(* CoDeSys 2.3.9.50 project: flat_v2.pro *)
(* Libraries: TcBABasic.lib 22.7.15 15:46:14, standard.lib 5.6.98 11:03:02, TcpIp.lib 9.1.14 13:33:22, TcBase.lib 14.5.09 11:14:08, TcSystem.lib 7.6.16 10:01:22, ModbusRTU.lib 13.5.15 12:38:16, TcIoFunctions.lib 27.1.17 16:22:22, COMlibV2.lb6 25.2.14 08:37:08, TcUtilities.lib 3.2.16 15:08:58 *)

(* Task configuration *)
TASK Standard (PRIORITY := 0, INTERVAL := T#50ms);
	MAIN
END_TASK

(* Global variable list: Global_Variables *)
VAR_GLOBAL


	Clear						: ClearComBuffer;
	MB							: ModbusRtuMaster_KL6x22B;
	TxBufferCom1				: ComBuffer;
	RxBufferCom1				: ComBuffer;
	SerialLineControlCom1			: SerialLineControl;
	ReceiveDataCom1			: ReceiveData;
	SendDataCom1				: SendData;
	Merc_address				: BYTE:=97;
	Sensor_CO2_high	 			: BYTE;	(*Старший байт датчика MH-Z19B*)
	Sensor_CO2_low 				: BYTE;	(*Младший байт датчика MH-Z19B*)
	iobroker						: iobroker_Struct;
	Modbus						: Modbus_Struct;
	Internal						: Internal_Struct;
(*
	MB_vars						: stMB;
	Mercury						: stMercury;
	iob_mqtt						: stIobroker;
*)
(*	Sensor_street_north_temp		: REAL;
	Sensor_sport_underfloor_temp	: REAL;
*)
	Sensor_control_temp			: WORD;
	Sensor_control_hum			: WORD;



	HW_temp_first_floor					AT %IW40:INT;	(* Датчик температуры 1 этаж *)
	HW_temp_second_floor				AT %IW42:INT;	(* Датчик температуры 2 этаж *)
	HW_temp_underfloor					AT %IW44:INT;	(* Датчик температуры подпол 1 этаж *)
	HW_temp_sport						AT %IW46:INT;	(* Датчик температуры спортзал *)

	HW_temp_sport_underfloor				AT %IW48:INT;	(* Датчик температуры подпол спортзал *)
	HW_temp_sauna						AT %IW50:INT;	(* Датчик температуры сауна*)
	HW_temp_street						AT %IW52:INT;	(* Датчик температуры улица *)
	HW_temp_vent						AT %IW54:INT;	(* Датчик температуры притока вентиляции *)

	HW_temp_balkon						AT %IW60:INT;	(* Датчик температуры  *)
	HW_temp_drovnik						AT %IW62:INT;	(* Датчик температуры *)
	HW_temp_sklad						AT %IW64:INT;	(* Датчик температуры  *)
	HW_temp_rezerv						AT %IW66:INT;	(* Датчик температуры  *)


	HW_PIR_terrasa						AT %IX56.0:BOOL;		(*PIR датчик терраса *)
	HW_PIR_zapad						AT %IX56.1:BOOL;		(*PIR датчик запад *)
	HW_PIR_vostok						AT %IX56.2:BOOL;		(*PIR датчик восток *)
	HW_PIR_sport						AT %IX56.3:BOOL;		(*PIR датчик спортзал *)

	HW_GERKON_drovnik					AT %IX56.4:BOOL;		(*Геркон дровник *)
	HW_GERKON_door					AT %IX56.5:BOOL;		(*Геркон дверь *)
	HW_sensor_smoke_1floor				AT %IX56.6:BOOL;		(*Датчик дыма 1 этаж *)
	HW_sensor_smoke_2_3floor			AT %IX56.7:BOOL;		(*Датчик дыма 2 этаж *)

	HW_button_light_garden				AT %IX57.0:BOOL;		(* Кнопка прожектор терраса  *)
	HW_sensor_smoke_sport				AT %IX57.1:BOOL;		(* Кнопка охрана  *)
	HW_button_vorota						AT %IX57.2:BOOL;		(* Кнопка открытия ворот  *)
	HW_button_kalitka					AT %IX57.3:BOOL;		(* Кнопка открытия калитки  *)

	HW_button_poliv_terrasa				AT %IX57.4:BOOL;		(* Кнопка полив терраса 2 часа  *)
	HW_button_poliv_zapad				AT %IX57.5:BOOL;		(* Кнопка полив запад  2 часа  *)
	HW_button_poliv_south				AT %IX57.6:BOOL;		(*  Кнопка полив юг  2 часа  *)
	HW_button_poliv_north					AT %IX57.7:BOOL;		(*  Кнопка полив север  2 часа  *)


	HW_sensor_supply					AT %IX58.0:BOOL;		(* Датчик напряжение  *)
	HW_GERKON_sklad					AT %IX58.1:BOOL;		(*Геркон *)
	HW_PIR_north_zapad					AT %IX58.2:BOOL;		(*PIR датчик  *)
	HW_PIR_north_vostok					AT %IX58.3:BOOL;		(*PIR датчик  *)


	HW_heat_first_floor					AT %QX0.0:BOOL;		(* Отопление 1 этаж *)
	HW_heat_second_floor				AT %QX0.1:BOOL;		(* Отопление 2 этаж *)
	HW_heat_sport						AT %QX0.2:BOOL;		(* Отопление спортзал *)
	HW_heat_underfloor					AT %QX0.3:BOOL;		(* Отопление подпол *)
	HW_heat_sauna						AT %QX0.4:BOOL;		(* Отопление сауна *)
	HW_heat_bathroom					AT %QX0.5:BOOL;		(* Отопление душевая *)
	HW_heat_pipe						AT %QX0.6:BOOL;		(* Отопление водопровод *)
	HW_vent_underfloor					AT %QX0.7:BOOL;		(* Вентиляция подпола *)

	HW_vorota							AT %QX1.0:BOOL;		(* Ворота *)
	HW_kalitka							AT %QX1.1:BOOL;		(* Калитка *)
	HW_pomp_house						AT %QX1.2:BOOL;		(* Насос водоснабжения дома *)
	HW_pomp_garden					AT %QX1.3:BOOL;		(* Насос полива *)
	HW_light_garden						AT %QX1.4:BOOL;		(* Прожектор двор *)
	HW_light_terrasa						AT %QX1.5:BOOL;		(* Свет терраса *)
	HW_light_rezerv						AT %QX1.6:BOOL;		(* Резервное освещение *)
	HW_switch_RS485					AT %QX1.7:BOOL:=TRUE;		(* RS485 line *)


	HW_vent_valve_input					AT %QX2.0:BOOL;		(* Клапан приточной вентиляции *)
	HW_vent_valve_output					AT %QX2.1:BOOL;		(* Клапан вытяжной вентиляции *)
	HW_trans_power						AT %QX2.2:BOOL;		(*Подача тока на трансформатор и реле ТЭН-а *)
	HW_vent_in_heat						AT %QX2.3:BOOL;		(* Подогрев притока - ТЭН *)
	HW_vent_in_heat_level				AT %QX2.4:BOOL;		(* Подогрев притока ночной режим   -5 К ТЭН *)
	HW_vent_in_trans_105_130				AT %QX2.5:BOOL:=FALSE;  (* Напряжение 110 или 130 В *)
	HW_vent_in_trans_160_220				AT %QX2.6:BOOL:=FALSE;  (* Напряжение 160 или 220 В *)
	HW_vent_in_trans_LO_HI				AT %QX2.7:BOOL:=FALSE;  (* Напряжение 110/130  или 160/220 В *)

	HW_poliv_terrasa						AT %QX3.0:BOOL;		(* полив терраса  *)
	HW_poliv_zapad						AT %QX3.1:BOOL;		(* полив запад   *)
	HW_poliv_south						AT %QX3.2:BOOL;		(* полив юг   *)
	HW_poliv_north						AT %QX3.3:BOOL;		(* полив север   *)
(*
	HW_level_light_1_floor					AT %QW4: WORD:=32767;	(* Уровень яркости света на 1 этаже *)
	HW_level_light_kitchen					AT %QW8: WORD:=32767;	(* Уровень яркости света на кухне *)
*)

END_VAR

(* Global variable list: TwinCAT_Configuration *)
(* Generated automatically by TwinCAT - (read only) *)
VAR_CONFIG
	MAIN.ToFromNovRam AT %QB56 : DataToFromNovram;	(*  ~ {LinkedWith:TIID^Device 2 (NOV/DP-RAM)^Outputs^Var4} *)
	.MB.InData AT %IB68 : MB_KL6inData22B;
	.MB.OutData AT %QB32 : MB_KL6outData22B;
END_VAR

(* Data type *)
TYPE DataToFromNovram :
STRUCT

	Target_CO2_mem					:		INT;
	First_floor_temp_target_mem		:		INT;
	Second_floor_temp_target_mem		:		INT;
	Sport_temp_target_mem			:		INT;
	Sauna_temp_target_mem			:		INT;
	Underfloor_temp_target_mem		:		INT;
	Underfloor_humidity_target_mem	:		INT;

	Pomp_house_mem				:		BOOL;
	Pomp_garden_mem				:		BOOL;

	Light_garden_mem				:		BOOL;

	Vent_mem						:		BOOL;
	Vent_heat_mem					:		INT;
	Vent_heat_level_mem				:		BOOL;

	Poliv_zapad_minutes				:		INT;
	Poliv_terrasa_minutes				:		INT;
	Poliv_south_minutes				:		INT;
	Poliv_north_minutes				:		INT;


END_STRUCT
END_TYPE

(* Data type *)
TYPE Internal_struct :
STRUCT
	Drovnik_temp					 :	REAL; 	(*12382*)			(* PT1000 *)
	Sklad_temp					 :	REAL; 	(*12384*)			(* PT1000 *)
	Rezerv_temp					 :	REAL; 	(*12386*)			(* PT1000 *)

	First_floor_temp 				:	REAL;	(*12288+100=12388*) (* PT1000 *)
	First_floor_hum 				:	REAL;	(*12390*)			(*SHT20		#1*)
	First_floor_CO2				:	REAL;	(*12392*)
	First_floor_temp_SHT20		:	REAL;	(*12394*)			(*SHT20		#1*)

	Second_floor_hum			:	REAL;	(*12396*)			(*SHT20		#2*)
	Second_floor_temp 			:	REAL;	(*12398*) 		(* PT1000 *)
	Second_floor_CO2 			:	REAL;	(*12400*)
	Sport_temp	 				:	REAL;	(*12402*)			(* PT1000 *)

	Sauna_temp	 				:	REAL;	(*12404*)			(* PT1000 *)
	Underfloor_temp				:	REAL;	(*12406*)			(* PT1000 *)
	Underfloor_hum				:	REAL;	(*12408*)			(*SHT20		#3*)
	Sport_underfloor_temp			:	REAL;	(*12410*)			(* PT1000 *)

	Sport_underfloor_hum			:	REAL;	(*12412*)			(*SHT20		#4*)
	Street_temp					:	REAL;	(*12414*)			(* PT1000 *)
	Vent_temp					:	REAL;	(*12416*)			(* PT1000 *)
	Sklad_temp_SHT20			:	REAL;	(*12418*)			(*SHT20		#5*)
	Sklad_hum					:	REAL;	(*12420*)			(*SHT20		#5*)
	Temp_vent_in				:	REAL;	(*12422*)			(* unused *)


	Uv1							:	REAL;	(*12424*)
	Uv2							:	REAL;	(*12426*)
	Uv3							:	REAL;	(*12428*)
	Pw1							:	REAL;	(*12430*)
	Pw2							:	REAL;	(*12432*)
	Pw3							:	REAL;	(*12434*)
	Pw_total						:	REAL;	(*12436*)
	Ia1							:	REAL;	(*12438*)
	Ia2							:	REAL;	(*12440*)
	Ia3							:	REAL;	(*12442*)
	E_T1						:	REAL;	(*12444*)
	E_T2						:	REAL; 	(*12288+158=12446*)

	Second_floor_temp_SHT20			:	REAL;	(*12448 *)		(*SHT20		#2*)
	Underfloor_temp_SHT20			:	REAL;	(*12450 *)		(*SHT20		#3*)
	Sport_underfloor_temp_SHT20		:	REAL;	(*12452 *)		(*SHT20		#4*)
	Street_temp_SHT20				:	REAL;	(*12454 *)		(*SHT20		#6*)
	Street_hum						:	REAL;	(*12456 *)		(*SHT20		#6*)

END_STRUCT
END_TYPE

(* Data type *)
TYPE iobroker_Struct  :
STRUCT
(*	Vent_status				: 	INT;
	Valve_status				: 	INT;
	First_floor_temp 			:	REAL;
	First_floor_temp_target 		:	INT;
	First_floor_hum 			:	REAL;
	First_floor_CO2			:	REAL;
	Kitchen_room_temp		:	REAL;
	Kitchen_room_hum		:	REAL;
	Second_floor_temp 		:	REAL;
	Second_floor_temp_target 	:	INT;
	Second_floor_CO2 		:	REAL;
	Sport_temp	 			:	REAL;
	Sport_temp_target			:	INT;
	Sauna_temp	 			:	REAL;
	Sauna_temp_target		:	INT;
	Underfloor_temp			:	REAL;
	Underfloor_temp_target	:	INT;
	Underfloor_humidity		:	REAL;
	Underfloor_humidity_target	:	INT;
	Sport_underfloor_temp		:	REAL;
	Sport_underfloor_hum		:	REAL;
	Street_temp				:	REAL;
	Vent_temp				:	REAL;
	Street_north_temp			:	REAL;
	Street_north_hum			:	REAL;
*)
	PIR_terrasa				:	BOOL:=TRUE;
	PIR_zapad				:	BOOL:=TRUE;
	PIR_vostok				:	BOOL:=TRUE;
	PIR_sport				:	BOOL:=TRUE;
	GERKON_drovnik			:	BOOL:=TRUE;
	Smoke					:	BOOL;
	Button_light_garden		:	BOOL;
	Light_garden				:	BOOL;
	Vorota_active				:	BOOL:=FALSE;
	Vorota_open_active		:	BOOL:=FALSE;
	Poliv_zapad				:	BOOL;
	Poliv_terrasa				:	BOOL;
	Poliv_south				:	BOOL;
	Poliv_north				:	BOOL;
(*
	Vent_input_level			:	INT;  (*  0-220 V  *)
	Vent_output_level			:	INT; (*0-100%*)
	Temp_vent_in			:	REAL;
	Vent_valve_status			:	INT;
	Security_status			:	BOOL;
	Target_CO2				:	INT;
	Vent						:	BOOL;
	Vent_underfloor			:	BOOL;
	Vent_out					:	BOOL;
	Vent_heat				:	INT;
	Vent_heat_level			:	BOOL;
	Vorota					:	BOOL;
	Vorota_open				:	BOOL;
	Kalitka					:	BOOL;
	
	Sensor_supply			:	BOOL;
	Pomp_house				:	BOOL;
	Pomp_garden			:	BOOL;
	Light_garden				:	BOOL;
	Poliv_zapad				:	BOOL;
	Poliv_terrasa				:	BOOL;
	Poliv_south				:	BOOL;
	Poliv_zapad_minutes		:	INT;
	Poliv_terrasa_minutes		:	INT;
	Poliv_south_minutes		:	INT;
	Uv1						:	REAL;
	Uv2						:	REAL;
	Uv3						:	REAL;
	Pw1						:	REAL;
	Pw2						:	REAL;
	Pw3						:	REAL;
	Pw_total					:	REAL;
	Ia1						:	REAL;
	Ia2						:	REAL;
	Ia3						:	REAL;
	E_T1					:	REAL;
	E_T2					:	REAL; (* 64 values*)
*)

(*	M1T1					:	DWORD:=0;
	M1T2					:	DWORD:=0; (* 66 values*)

	M2T1					:	DWORD:=0; (* 67 values*)
	M2T2					:	DWORD:=0;
	M3T1					:	DWORD:=0;
	M3T2					:	DWORD:=0;
	M4T1					:	DWORD:=0; (* 70 values*)
	M4T2					:	DWORD:=0;
	M5T1					:	DWORD:=0;
	M5T2					:	DWORD:=0;
	M6T1					:	DWORD:=0;
	M6T2					:	DWORD:=0;
	M7T1					:	DWORD:=0;
	M7T2					:	DWORD:=0;
	M8T1					:	DWORD:=0;
	M8T2					:	DWORD:=0;
	M9T1					:	DWORD:=0;
	M9T2					:	DWORD:=0;
	M10T1					:	DWORD:=0;
	M10T2					:	DWORD:=0;
	M11T1					:	DWORD:=0;
	M11T2					:	DWORD:=0;
	M12T1					:	DWORD:=0;
	M12T2					:	DWORD:=0;   (* 86 values*)
*)

END_STRUCT
END_TYPE

(* Data type *)
TYPE Modbus_struct :
STRUCT
	Vent_status					AT %MB100	:	INT;		(*12288+50=12338*)
	Valve_status					AT %MB102	: 	INT;		(*12339*)
	First_floor_temp_target 			AT %MB104	:	INT;		(*12340*)
	Second_floor_temp_target 		AT %MB106	:	INT;		(*12341*)
	Sport_temp_target				AT %MB108	:	INT;		(*12342*)
	Sauna_temp_target			AT %MB110	:	INT;		(*12343*)
	Underfloor_temp_target		AT %MB112	:	INT;		(*12344*)
	Underfloor_humidity_target		AT %MB114	:	INT;		(*12345*)
	PIR_terrasa					AT %MB116	:	BOOL:=TRUE;	(*12346*)
	PIR_zapad					AT %MB118	:	BOOL:=TRUE;	(*12347*)
	PIR_vostok					AT %MB120	:	BOOL:=TRUE;	(*12348*)
	PIR_sport					AT %MB122	:	BOOL:=TRUE;	(*12349*)
	GERKON_drovnik				AT %MB124	:	BOOL:=TRUE;	(*12288+62=12350*)

	Vent_input_level				AT %MB126	:	INT; 			 (*12351			*  0-220 V  *)
	Vent_output_level				AT %MB128	:	INT; 			(*12352			0-100%*)
	Vent_valve_status				AT %MB130	:	INT;		(*12353*)
	Target_CO2					AT %MB132	:	INT;		(*12354*)
	Security_status				AT %MB134	:	BOOL;	(*12355*)
	Vent							AT %MB136	:	BOOL;	(*12356*)
	Vent_underfloor				AT %MB138	:	BOOL;	(*12357*)
	Vent_out						AT %MB140	:	BOOL;	(*12358*)
	Vent_heat					AT %MB142	:	INT;		(*12359*)
	Vent_heat_level				AT %MB144	:	BOOL;	(*12360*)
	Vorota						AT %MB146	:	BOOL;	(*12361*)
	Vorota_open					AT %MB148	:	BOOL;	(*12362*)
	Kalitka						AT %MB150	:	BOOL;	(*12363*)
(*
	Smoke						AT %MB152	:	BOOL;	(*12364*)
*)
	Sensor_supply				AT %MB154	:	BOOL;	(*12365*)
	Pomp_house					AT %MB156	:	BOOL;	(*12366*)
	Pomp_garden				AT %MB158	:	BOOL;	(*12367*)
	Light_garden					AT %MB160	:	BOOL;	(*12368*)
	Poliv_zapad					AT %MB162	:	BOOL;	(*12369*)
	Poliv_terrasa					AT %MB164	:	BOOL;	(*12370*)
	Poliv_south					AT %MB166	:	BOOL;	(*12371*)
	Poliv_zapad_minutes			AT %MB168	:	INT;		(*12372*)
	Poliv_terrasa_minutes			AT %MB170	:	INT;		(*12373*)
	Poliv_south_minutes			AT %MB172	:	INT;		(*12288 +86=  12374*)
	Poliv_north_minutes			AT %MB174	:	INT	;	(*12375 *)
	Poliv_north					AT %MB176	:	BOOL;	(*12376*)






	Drovnik_temp					AT %MW188 :	REAL; 	(*12382*)			(* PT1000 *)
	Sklad_temp					AT %MW192 :	REAL; 	(*12384*)			(* PT1000 *)
	Rezerv_temp					AT %MW196 :	REAL; 	(*12386*)			(* PT1000 *)

	First_floor_temp 				AT %MW200	:	REAL;	(*12288+100=12388*) (* PT1000 *)
	First_floor_hum 				AT %MW204	:	REAL;	(*12390*)			(*SHT20		#1*)
	First_floor_CO2				AT %MW208	:	REAL;	(*12392*)
	First_floor_temp_SHT20		AT %MW212	:	REAL;	(*12394*)			(*SHT20		#1*)

	Second_floor_hum			AT %MW216	:	REAL;	(*12396*)			(*SHT20		#2*)
	Second_floor_temp 			AT %MW220	:	REAL;	(*12398*) 		(* PT1000 *)
	Second_floor_CO2 			AT %MW224	:	REAL;	(*12400*)
	Sport_temp	 				AT %MW228	:	REAL;	(*12402*)			(* PT1000 *)

	Sauna_temp	 				AT %MW232	:	REAL;	(*12404*)			(* PT1000 *)
	Underfloor_temp				AT %MW236	:	REAL;	(*12406*)			(* PT1000 *)
	Underfloor_hum				AT %MW240	:	REAL;	(*12408*)			(*SHT20		#3*)
	Sport_underfloor_temp			AT %MW244	:	REAL;	(*12410*)			(* PT1000 *)

	Sport_underfloor_hum			AT %MW248	:	REAL;	(*12412*)			(*SHT20		#4*)
	Street_temp					AT %MW252	:	REAL;	(*12414*)			(* PT1000 *)
	Vent_temp					AT %MW256	:	REAL;	(*12416*)			(* PT1000 *)
	Sklad_temp_SHT20			AT %MW260	:	REAL;	(*12418*)			(*SHT20		#5*)
	Sklad_hum					AT %MW264	:	REAL;	(*12420*)			(*SHT20		#5*)
	Temp_vent_in				AT %MW268	:	REAL;	(*12422*)			(* unused *)


	Uv1							AT %MW272	:	REAL;	(*12424*)
	Uv2							AT %MW276	:	REAL;	(*12426*)
	Uv3							AT %MW280	:	REAL;	(*12428*)
	Pw1							AT %MW284	:	REAL;	(*12430*)
	Pw2							AT %MW288	:	REAL;	(*12432*)
	Pw3							AT %MW292	:	REAL;	(*12434*)
	Pw_total						AT %MW296	:	REAL;	(*12436*)
	Ia1							AT %MW300	:	REAL;	(*12438*)
	Ia2							AT %MW304	:	REAL;	(*12440*)
	Ia3							AT %MW308	:	REAL;	(*12442*)
	E_T1						AT %MW312	:	REAL;	(*12444*)
	E_T2						AT %MW316	:	REAL; 	(*12288+158=12446*)

	Second_floor_temp_SHT20		AT %MW320	:	REAL;	(*12448 *)		(*SHT20		#2*)
	Underfloor_temp_SHT20		AT %MW324	:	REAL;	(*12450 *)		(*SHT20		#3*)
	Sport_underfloor_temp_SHT20	AT %MW328	:	REAL;	(*12452 *)		(*SHT20		#4*)
	Street_temp_SHT20			AT %MW332	:	REAL;	(*12454 *)		(*SHT20		#6*)
	Street_hum					AT %MW336	:	REAL;	(*12456 *)		(*SHT20		#6*)


	Smoke_1floor					AT %MB400	:	BOOL;	(*12288+200=12488*)
	Smoke_2_3floor				AT %MB402	:	BOOL;	(*12489*)
	Smoke_sport					AT %MB404	:	BOOL;	(*12490*)
	Rezerv_2					AT %MB406	:	BOOL;	(*12491*)
	PIR_north_zapad				AT %MB408	:	BOOL;	(*12492*)
	PIR_north_vostok				AT %MB410	:	BOOL;	(*12493*)
	Gerkon_sklad				AT %MB412	:	BOOL;	(*12494*)
	Gerkon_door					AT %MB414	:	BOOL;	(*12495*)
	Light_reserv					AT %MB416	:	BOOL;	(*12496*)
	Light_reserv_manual			AT %MB418	:	INT;		(*12497*)
	Supply_akb					AT %MB420	:	REAL;	(*12498*)
	Security_delay				AT %MB424	:	INT;		(*12500*)
	Balkon_temp					AT %MW428 :	REAL; 	(*12502*)			(* PT1000 *)

	Poliv_zapad_minutes_est		AT %MB500	:	INT;		(*12288+250=12538*)
	Poliv_terrasa_minutes_est		AT %MB502	:	INT;		(*12539*)
	Poliv_south_minutes_est		AT %MB504	:	INT;		(*12540*)
	Poliv_north_minutes_est		AT %MB506	:	INT	;	(*12541 *)

	Kitchen_room_CO2			AT %MB508	:	INT;

	M1T1					AT %MB600	:	REAL;
	M1T2					AT %MB604	:	REAL;
	M2T1					AT %MB608	:	REAL;
	M2T2					AT %MB612	:	REAL;
	M3T1					AT %MB616	:	REAL;
	M3T2					AT %MB620	:	REAL;
	M4T1					AT %MB624	:	REAL;
	M4T2					AT %MB628	:	REAL;
	M5T1					AT %MB632	:	REAL;
	M5T2					AT %MB636	:	REAL;
	M6T1					AT %MB640	:	REAL;
	M6T2					AT %MB644	:	REAL;
	M7T1					AT %MB648	:	REAL;
	M7T2					AT %MB652	:	REAL;
	M8T1					AT %MB656	:	REAL;
	M8T2					AT %MB660	:	REAL;
	M9T1					AT %MB664	:	REAL;
	M9T2					AT %MB668	:	REAL;
	M10T1					AT %MB672	:	REAL;
	M10T2					AT %MB676	:	REAL;
	M11T1					AT %MB680	:	REAL;
	M11T2					AT %MB684	:	REAL;
	M12T1					AT %MB688	:	REAL;
	M12T2					AT %MB692	:	REAL;


END_STRUCT
END_TYPE

(* Data type *)
(* @NESTEDCOMMENTS := 'Yes' *)
(* @PATH := '' *)
(* @OBJECTFLAGS := '0, 8' *)
TYPE ST_MqttReceivedPublishTelegram :
STRUCT
	sTopic		: STRING[255];
	sValue		: STRING[255];
	bHasData	: BOOL;
END_STRUCT
END_TYPE
(* @END_DECLARATION := '0' *)

(* Data type *)
(* @NESTEDCOMMENTS := 'Yes' *)
(* @PATH := '' *)
(* @OBJECTFLAGS := '0, 8' *)
TYPE ST_MqttSettings :
STRUCT
	(* informations *)
	sMqttClientId	: STRING[23];
	sMqttUserId	: STRING[25];
	sMqttPassword	: STRING[25];
	sMqttBrokerIP	: STRING[15];
	nMqttBrokerPort	: UDINT := 1883;

	(* state *)
	bSocketConnection	: BOOL := FALSE;
	bConnected			: BOOL := FALSE;
	bConnectPackageSent	: BOOL := FALSE;
	bDisconnect			: BOOL := FALSE;
	bError				: BOOL := FALSE;
	bValidConnection	: BOOL := FALSE;
	bActive				: BOOL := FALSE;
	wPackageIdentifier	: WORD := 1;
	hSocket				: T_HSOCKET;
	tonSendPingReq		: TON;

	(* send *)
	stMqttSendTelegram			: ST_MqttTelegram;
	stMqttLastSendTelegram		: ST_MqttTelegram;

	(* receive *)
	stMqttReceivedTelegram			: ST_MqttTelegram;
	stMqttLastReceivedTelegram		: ST_MqttTelegram;
	stMqttReceivedPublishTelegram	: ST_MqttReceivedPublishTelegram;

	(* settings internal *)
	iTelegramSize	: INT := 544;
	usKeepAliveTime	: USINT := 60; (* seconds *)

END_STRUCT
END_TYPE
(* @END_DECLARATION := '0' *)

(* Data type *)
(* @NESTEDCOMMENTS := 'Yes' *)
(* @PATH := '' *)
(* @OBJECTFLAGS := '0, 8' *)
TYPE ST_MqttTelegram :
STRUCT
	arMqttData 	: ARRAY[0..544] OF BYTE;
	nDataLength	: UDINT := 0;
END_STRUCT
END_TYPE
(* @END_DECLARATION := '0' *

(* Data type *)
TYPE stIobroker :
STRUCT

	Control_hum					:	REAL;
	Control_temp					:	REAL;
	Control_hum2					:	REAL;
	Control_temp2				:	REAL;

END_STRUCT
END_TYPE

(* Data type *)
TYPE stMB :
STRUCT

	M1T1							AT %MW0	:REAL;  	(* modbus address 12288 *)
	M1T2							AT %MW4	:REAL;	(* 12290 *)
	M2T1							AT %MW8	:REAL;	(* 12292 *)
	M2T2							AT %MW12	:REAL;	 (* 12294 *)
	M3T1							AT %MW16	:REAL;	 (* 12296 *)
	M3T2							AT %MW20	:REAL;	 (* 12298 *)
	M4T1							AT %MW24	:REAL;	 (* 12300 *)
	M4T2							AT %MW28	:REAL;	 (* 12302 *)
	M5T1							AT %MW32	:REAL;	 (* 12304 *)
	M5T2							AT %MW36	:REAL;	 (* 12306 *)
	M6T1							AT %MW40	:REAL;	 (* 12308 *)
	M6T2							AT %MW44	:REAL;	(* 12310 *)
	M7T1							AT %MW48	:REAL;	 (* 12312 *)
	M7T2							AT %MW52	:REAL;	 (* 12314 *)
	M8T1							AT %MW56	:REAL;	 (* 12316 *)
	M8T2							AT %MW60	:REAL;	(* 12318 *)
	M9T1							AT %MW64	:REAL;	(* 12320 *)
	M9T2							AT %MW68	:REAL;	(* 12322 *)
	M10T1							AT %MW72	:REAL;	(* 12324 *)
	M10T2							AT %MW76	:REAL;	(* 12326 *)
	M11T1							AT %MW80	:REAL;	(* 12328 *)
	M11T2							AT %MW84	:REAL;	(* 12330 *)
	M12T1							AT %MW88	:REAL;	(* 12332 *)
	M12T2							AT %MW92	:REAL;	(* 12334 *)

END_STRUCT
END_TYPE

(* Data type *)
TYPE stMercury :
STRUCT

	M1T1					:	REAL;
	M1T2					:	REAL;
	M2T1					:	REAL;
	M2T2					:	REAL;
	M3T1					:	REAL;
	M3T2					:	REAL;
	M4T1					:	REAL;
	M4T2					:	REAL;
	M5T1					:	REAL;
	M5T2					:	REAL;
	M6T1					:	REAL;
	M6T2					:	REAL;
	M7T1					:	REAL;
	M7T2					:	REAL;
	M8T1					:	REAL;
	M8T2					:	REAL;
	M9T1					:	REAL;
	M9T2					:	REAL;
	M10T1					:	REAL;
	M10T2					:	REAL;
	M11T1					:	REAL;
	M11T2					:	REAL;
	M12T1					:	REAL;
	M12T2					:	REAL;

END_STRUCT
END_TYPE

(* POU MAIN, ST *)
PROGRAM MAIN
VAR
	ToFromNovRam			AT %Q*:DataToFromNovram;
	INITVAR					: BOOL:=FALSE;




END_VAR
IF (INITVAR=FALSE) THEN

	(* START RESTORE VARS FROM MEMORY AFTER REBOOT/RESET/LOST POWER *)

	Modbus.Target_CO2				:=	ToFromNovRam.Target_CO2_mem;
	Modbus.First_floor_temp_target		:=	ToFromNovRam.First_floor_temp_target_mem;
	Modbus.Second_floor_temp_target	:=	ToFromNovRam.Second_floor_temp_target_mem;
	Modbus.Sport_temp_target			:=	ToFromNovRam.Sport_temp_target_mem;
	Modbus.Sauna_temp_target		:=	ToFromNovRam.Sauna_temp_target_mem;

	Modbus.Underfloor_temp_target		:=	ToFromNovRam.Underfloor_temp_target_mem;
	Modbus.Underfloor_humidity_target	:=	ToFromNovRam.Underfloor_humidity_target_mem;

	Modbus.Vent						:=	ToFromNovRam.Vent_mem;
	Modbus.Vent_heat				:=	ToFromNovRam.Vent_heat_mem;
	Modbus.Vent_heat_level			:=	ToFromNovRam.Vent_heat_level_mem;

	Modbus.Pomp_house				:=	ToFromNovRam.Pomp_house_mem;
	Modbus.Pomp_garden				:=	ToFromNovRam.Pomp_garden_mem;
	Modbus.Light_garden				:=	ToFromNovRam.Light_garden_mem;

	Modbus.Poliv_zapad_minutes		:=	ToFromNovRam.Poliv_zapad_minutes;
	Modbus.Poliv_terrasa_minutes		:=	ToFromNovRam.Poliv_terrasa_minutes;
	Modbus.Poliv_south_minutes		:=	ToFromNovRam.Poliv_south_minutes;
	Modbus.Poliv_north_minutes		:=	ToFromNovRam.Poliv_north_minutes;

	(* END RESTORE VARS FROM MEMORY AFTER REBOOT/RESET/LOST POWER *)

	INITVAR:=TRUE;
ELSE
	(*START SAVE VARS to PERSISTENT MEMORY*)
	ToFromNovRam.Target_CO2_mem					:=	Modbus.Target_CO2;
	ToFromNovRam.First_floor_temp_target_mem			:=	Modbus.First_floor_temp_target;
	ToFromNovRam.Second_floor_temp_target_mem		:=	Modbus.Second_floor_temp_target;
	ToFromNovRam.Sport_temp_target_mem			:=	Modbus.Sport_temp_target;
	ToFromNovRam.Sauna_temp_target_mem			:=	Modbus.Sauna_temp_target;

	ToFromNovRam.Underfloor_temp_target_mem		:=	Modbus.Underfloor_temp_target;
	ToFromNovRam.Underfloor_humidity_target_mem		:=	Modbus.Underfloor_humidity_target;

	ToFromNovRam.Vent_mem						:=	Modbus.Vent;
	ToFromNovRam.Vent_heat_mem					:=	Modbus.Vent_heat;
	ToFromNovRam.Vent_heat_level_mem				:=	Modbus.Vent_heat_level;

	ToFromNovRam.Pomp_house_mem				:=	Modbus.Pomp_house;
	ToFromNovRam.Pomp_garden_mem			:=	Modbus.Pomp_garden;
	ToFromNovRam.Light_garden_mem				:=	Modbus.Light_garden;


	ToFromNovRam.Poliv_zapad_minutes			:=	Modbus.Poliv_zapad_minutes;
	ToFromNovRam.Poliv_terrasa_minutes			:=	Modbus.Poliv_terrasa_minutes;
	ToFromNovRam.Poliv_south_minutes			:=	Modbus.Poliv_south_minutes;
	ToFromNovRam.Poliv_north_minutes			:=	Modbus.Poliv_north_minutes;

	(*END SAVE VARS to PERSISTENT MEMORY*)


	Sensors;						(* Аналогвые датчики на шине KL *)
	Security_new;						(* Мониторинг датчиков охраны *)
	RS485read;					(* Опрос устройств на шине RS485 *)
(*	Mqtt;	*)					(* MQTT *)
	Thermocontrol;				(* Термостат*)
	VentControl;					(* Глобальный контроль вентустановки*)
	VentPower;					(* Авторегулировка мощности вентустановки по датчикам CO2*)
	Poliv;						(* Таймеры зонального полива *)
	Power_act;					(*Контроль резервного освещения*)



(* Прямое присовение виртуальных переменных к переменным, жестко привязаным к физ. портам. Частота обновления= циклу ПЛК (50 мсек) : *)
	HW_pomp_house				:=	Modbus.Pomp_house;
	Modbus.Sensor_supply		:=	HW_sensor_supply;
	HW_vent_underfloor			:=	Modbus.Vent_underfloor;

	HW_kalitka					:=	Modbus.Kalitka;
	iobroker.button_light_garden	:=	HW_button_light_garden;
	HW_light_garden				:=	Modbus.Light_garden;
	iobroker.Light_garden			:=	Modbus.Light_garden;


	Buttons;						(*Обработка нажатия кнопок *)

END_IF
END_PROGRAM

(* POU Sensors, ST *)
PROGRAM Sensors
VAR
(*	Period_sensors_read		: INT:=30; *) (* Частота присвоения значений аналоговых температурных датчиков с модулей KL, секунды *)
	Timer					: TON;
	TimerQ					: BOOL;
	tTimerValue				: TIME:=t#30s; (* Частота присвоения значений аналоговых температурных датчиков с модулей KL, секунды *)
END_VAR
Timer();

(* tTimerValue := DINT_TO_TIME(Period_sensors_read*1000); *)

	Timer(IN:=NOT TimerQ , PT:=tTimerValue , Q=>TimerQ , ET=> );
	IF timer.q THEN

		Modbus.First_floor_temp		:=	INT_TO_REAL(HW_temp_first_floor)/10;
		Modbus.Second_floor_temp	:=	INT_TO_REAL(HW_temp_second_floor)/10;
		Modbus.Sauna_temp			:=	INT_TO_REAL(HW_temp_sauna)/10;
		Modbus.Sport_temp			:=	INT_TO_REAL(HW_temp_sport)/10;

		Modbus.Underfloor_temp		:=	INT_TO_REAL(HW_temp_underfloor)/10;
		Modbus.Sport_underfloor_temp	:=	INT_TO_REAL(HW_temp_sport_underfloor)/10;
		Modbus.Street_temp			:=	INT_TO_REAL(HW_temp_street)/10;
		Modbus.Vent_temp			:=	INT_TO_REAL(HW_temp_vent)/10;

		Modbus.Balkon_temp			:=	INT_TO_REAL(HW_temp_balkon)/10;
		Modbus.Drovnik_temp			:=	INT_TO_REAL(HW_temp_drovnik)/10;
		Modbus.Sklad_temp			:= 	INT_TO_REAL(HW_temp_sklad)/10;

	END_IF
END_PROGRAM

(* POU Security_new, ST *)
PROGRAM Security_new
VAR
(*	TRIG_PIR_terrasa			:	F_TRIG;
	TRIG_PIR_zapad			:	F_TRIG;
	TRIG_PIR_vostok			:	F_TRIG;
	TRIG_PIR_sport			:	F_TRIG;
	TRIG_GERKON_drovnik	:	F_TRIG;
	TRIG_sensor_smoke_1floor:	F_TRIG;

	trig_mem_terrasa				:	BOOL:=FALSE;
	trig_mem_zapad				:	BOOL:=FALSE;
	trig_mem_vostok				:	BOOL:=FALSE;
	trig_mem_sport				:	BOOL:=FALSE;
	trig_mem_drovnik				:	BOOL:=FALSE;
	trig_mem_sensor_smoke_1floor	:	BOOL:=FALSE;
*)
END_VAR
iobroker.PIR_terrasa			 :=HW_PIR_terrasa;
iobroker.PIR_zapad			 :=HW_PIR_zapad;
iobroker.PIR_vostok 			 :=HW_PIR_vostok;
iobroker.PIR_sport			 :=HW_PIR_sport;
iobroker.GERKON_drovnik		 :=HW_GERKON_drovnik;

Modbus.Smoke_1floor				 :=HW_sensor_smoke_1floor;
Modbus.Smoke_2_3floor			 :=HW_sensor_smoke_2_3floor;
Modbus.Smoke_sport				 :=HW_sensor_smoke_sport;


Modbus.PIR_terrasa			 :=HW_PIR_terrasa;
Modbus.PIR_zapad			 :=HW_PIR_zapad;
Modbus.PIR_vostok 			 :=HW_PIR_vostok;
Modbus.PIR_sport				 :=HW_PIR_sport;
Modbus.PIR_north_zapad		 :=HW_PIR_north_zapad;
Modbus.PIR_north_vostok		 :=HW_PIR_north_vostok;

Modbus.GERKON_door		 :=HW_GERKON_door;
Modbus.GERKON_drovnik		 :=HW_GERKON_drovnik;
Modbus.GERKON_sklad		 :=HW_GERKON_sklad;



(* Modbus.Smoke				 :=HW_sensor_smoke_1floor; *)
END_PROGRAM

(* POU RS485read, ST *)
PROGRAM RS485read
VAR
(*	Period_vent_switch	: INT:=180; *)
	CO2_period			: TIME;
	tTimerValue			: TIME	:=	t#180s; (* Период опроса RS485*)

	password_1				: ARRAY [1..6] OF BYTE:=6(1); (* пароль к меркуриям, по умолчанию 6 единиц*)
	crctest					: WORD;
	arrReceive				: ARRAY[1..22] OF BYTE;
	arrSend					: ARRAY[1..22] OF BYTE;

	MBdata					 : ARRAY [1..2] OF INT;
	FtrigBusy				: F_TRIG;
	timeoutvalue				: TIME := T#1000ms;		(* timeout while waiting for an answer of the modbus slave *)
	state					: INT;
	busy					: BOOL;
	LastErrorstate				: INT;
	LastModbusError			: ST_ModbusErrorDiagnostics;
	CounterError				: DINT;
	CounterSuccess			: DINT;
	Timer1					: TON;
	Timer1Q					: BOOL;
	Timer_day				:TON;
	Timer_dayQ				:BOOL;
	Timer_CO2				:TON;
(*	Timer_CO2Q				:BOOL; *)

	tmCheck					:TON;
	i,k,l,m,t					: INT:=1;


	sensors_SHT20_v1_id			: ARRAY[1..2] OF BYTE:=16#05, 16#0F;
	sensors_SHT20_v1_hum		: ARRAY[1..2] OF REAL:=2(0);
	sensors_SHT20_v1_temp		: ARRAY[1..2] OF REAL:=2(0);

	sensors_SHT20_v2_id			: ARRAY[1..4] OF BYTE:= 16#07, 16#08, 16#09,16#0A;
	sensors_SHT20_v2_hum		: ARRAY[1..4] OF REAL:=4(0);
	sensors_SHT20_v2_temp		: ARRAY[1..4] OF REAL:=4(0);


	sensors_CO2_id				: ARRAY[1..1] OF BYTE:=16#68;
	sensors_CO2_ppm			: ARRAY[1..1] OF INT;

	energyMT					: ARRAY[1..12,1..2] OF REAL;

	get_co2_mh_z19b_1floor	: FB_GET_CO2_MH_Z19B;
	get_co2_mh_z19b_2floor	: FB_GET_CO2_MH_Z19B;
	get_supply				: FB_GET_SUPPLY;
	get_current				: FB_GET_CURRENT;
	get_power				: FB_GET_POWER;
	get_energy_E_T1			: FB_GET_ENERGY;
	get_energy_E_T2			: FB_GET_ENERGY;

	get_energy_MT			: FB_GET_ENERGY;



	get_co2_mh_z19b_1floor_done	: BOOL;
	get_co2_mh_z19b_2floor_done	: BOOL;
	get_supply_done			: BOOL;
	get_current_done			: BOOL;
	get_power_done			: BOOL;

	get_energy_E_T1_done	: BOOL;
	get_energy_E_T2_done	: BOOL;
	get_energy_MT_done		: BOOL;

END_VAR
tmCheck();
Timer_day();
Timer_CO2();


IF (Modbus.Security_status = TRUE) THEN
	CO2_period	:= T#30m;
ELSE
	CO2_period 	:= T#2m;
END_IF


CASE state OF
	0:
		MB.ReadRegs(Execute:= FALSE);
		state := 1;


1:
	Clear(Buffer := RxBufferCom1);
		MB.ReadRegs(
			UnitID:= sensors_SHT20_v1_id[i],
			Quantity:= 2,
			MBAddr:= 0,
			cbLength:= 6,
			pMemoryAddr:= ADR(MBdata),
			Execute:= TRUE,
			Timeout:= timeoutvalue,
			Busy => busy,
		);
		IF NOT busy THEN
			IF (mb.Error = FALSE ) THEN
				sensors_SHT20_v1_temp[i]:=INT_TO_REAL(MBdata[1])/10;
				sensors_SHT20_v1_hum[i]:=INT_TO_REAL(MBdata[2])/10;
			END_IF
			i:=i+1;
			MB.ReadRegs(Execute:= FALSE);
			IF (i>2 )	THEN
				i:=1;
				Internal.First_floor_temp_SHT20		:=	sensors_SHT20_v1_temp[1];
				Internal.First_floor_hum				:=	sensors_SHT20_v1_hum[1];
				Internal.Street_temp_SHT20			:=	sensors_SHT20_v1_temp[2];
				Internal.Street_hum				:=	sensors_SHT20_v1_hum[2];
				Modbus.First_floor_temp_SHT20	:=	(sensors_SHT20_v1_temp[1]);
				Modbus.First_floor_hum			:=	(sensors_SHT20_v1_hum[1]);
				Modbus.Street_temp_SHT20		:=	(sensors_SHT20_v1_temp[2]);
				Modbus.Street_hum				:=	(sensors_SHT20_v1_hum[2]);
				state :=2;
			ELSE
				state :=1;
			END_IF

		END_IF

2:

		MB.ReadInputRegs(
			UnitID:= sensors_SHT20_v2_id[l],
			Quantity:= 2,
			MBAddr:= 1,
			cbLength:= 6,
			pMemoryAddr:= ADR(MBdata),
			Execute:= TRUE,
			Timeout:= timeoutvalue,
			Busy => busy,
		);
		IF NOT busy THEN
			IF (mb.Error = FALSE ) THEN
				sensors_SHT20_v1_temp[l]:=INT_TO_REAL(MBdata[1])/10;
				sensors_SHT20_v1_hum[l]:=INT_TO_REAL(MBdata[2])/10;
			END_IF
			l:=l+1;
			MB.ReadRegs(Execute:= FALSE);
			IF (l>4 )	THEN
				l:=1;
				Internal.Underfloor_temp_SHT20				:=	sensors_SHT20_v2_temp[1];
				Internal.Underfloor_hum					:=	sensors_SHT20_v2_hum[1];
				Internal.Sport_underfloor_temp_SHT20		:=	sensors_SHT20_v2_temp[2];
				Internal.Sport_underfloor_hum				:=	sensors_SHT20_v2_hum[2];
				Internal.Second_floor_temp_SHT20			:=	sensors_SHT20_v2_temp[3];
				Internal.Second_floor_hum					:=	sensors_SHT20_v2_hum[3];
				Internal.Sklad_temp_SHT20					:=	sensors_SHT20_v2_temp[4];
				Internal.Sklad_hum						:=	sensors_SHT20_v2_hum[4];


				Modbus.Underfloor_temp_SHT20			:=	(sensors_SHT20_v2_temp[1]);
				Modbus.Underfloor_hum					:=	(sensors_SHT20_v2_hum[1]);
				Modbus.Sport_underfloor_temp_SHT20		:=	(sensors_SHT20_v2_temp[2]);
				Modbus.Sport_underfloor_hum				:=	(sensors_SHT20_v2_hum[2]);
				Internal.Second_floor_temp_SHT20			:=	sensors_SHT20_v2_temp[3];
				Internal.Second_floor_hum					:=	sensors_SHT20_v2_hum[3];
				Internal.Sklad_temp_SHT20					:=	sensors_SHT20_v2_temp[4];
				Internal.Sklad_hum						:=	sensors_SHT20_v2_hum[4];

				state :=3;
			ELSE
				state :=2;
			END_IF

		END_IF



3:
		MB.ReadInputRegs(
			UnitID:=sensors_CO2_id[k], (* station address *)
			Quantity:= 1,
			MBAddr:= 3,
			cbLength:= 4,
			pMemoryAddr:= ADR(MBdata),
			Execute:= TRUE,
			Timeout:= timeoutvalue,
			Busy => busy	);
		IF NOT busy THEN
			IF (mb.Error = FALSE ) THEN
				sensors_CO2_ppm[k]	:=	(MBdata[1]);
			END_IF
			k:=k+1;
			MB.ReadRegs(Execute:= FALSE);
			IF (k>1 )	THEN
				k:=1;

				Modbus.Kitchen_room_CO2		:=	(sensors_CO2_ppm[1]);

				state :=5;
			ELSE
				state :=3;
			END_IF
		END_IF


5:

		tmCheck(in:=FALSE);
		tmCheck(in:=TRUE,pt:=t#2s);
		get_co2_mh_z19b_2floor_done := FALSE;
		get_co2_mh_z19b_2floor( co2=>Modbus.Second_Floor_CO2, done=>get_co2_mh_z19b_2floor_done);
		IF get_co2_mh_z19b_2floor_done = TRUE THEN
			state:=105;
		ELSIF tmcheck.Q THEN
			 state:=105;
		END_IF


105: (*открываем канал*)


	Clear(Buffer := RxBufferCom1);
	arrSend[1]:=Merc_address;
	arrSend[2]:=1; (*код доступа*)
	arrSend[3]:=1; (*Уровень доступа*)

	MEMCPY(ADR(arrSend)+3,ADR(password_1),6); (*пароль*)
	crctest:=F_CRC16(ADR(arrSend),9); (*расчет контрольной суммы*)
	MEMCPY(ADR(arrSend)+9,ADR(crctest),SIZEOF(crctest)); (*прибавление контрольной суммы к запросу*)
	SendDataCom1(pSendData:=ADR(arrSend),Length:=11,TXBuffer:=TxBufferCom1,Busy=>,Error=>);
	tmCheck(in:=FALSE); tmCheck(in:=TRUE,pt:=t#2s); 	(*запуск таймера проверки - потеря связи\обрыв кабеля*)
	state:=106;

106: (*ответ*)
	ReceiveDataCom1(pPrefix:=,LenPrefix:=,pSuffix:=,LenSuffix:=,
	pReceiveData:=ADR(arrReceive),SizeReceiveData:=4,
	Timeout:=t#2s,Reset:=,
	RXbuffer:=RxBufferCom1,
	DataReceived=>,busy=>,Error=>,RxTimeout=>,LenReceiveData=>);
	IF ReceiveDataCom1.Error <> 0 THEN
		state:=888;
	END_IF
	IF receiveDataCom1.DataReceived THEN
		state:=107;
	ELSIF tmcheck.Q THEN
		state:=888;
	END_IF
107: (*проверка ответа*)

	IF arrReceive[1] = Merc_address THEN
		state:= 108;
	ELSE
		state:=888;
	END_IF



108:
		tmCheck(in:=FALSE);
		tmCheck(in:=TRUE,pt:=t#2s);
		get_supply_done := FALSE;
		get_supply( byte1:=16#8, byte2:=16#16, byte3:=16#11,  supply1=>Modbus.UV1,supply2=>Modbus.UV2,supply3=>Modbus.UV3, done=>get_supply_done);
		IF get_supply_done = TRUE THEN
			state:=109;
		ELSIF tmcheck.Q THEN
			 state:=888;
		END_IF

 (*запрос на чтение тока  на всех фазах
--------------------------------------------------------------------------------------------------------------------------------------------------------------------
*)
109:
		tmCheck(in:=FALSE);
		tmCheck(in:=TRUE,pt:=t#2s);
		get_current_done := FALSE;
		get_current(byte1:=16#8, byte2:=16#16, byte3:=16#21,  current1=>Modbus.Ia1,current2=>Modbus.Ia2,current3=>Modbus.Ia3, done=>get_current_done);
		IF get_current_done = TRUE THEN
			state:=110;
		ELSIF tmcheck.Q THEN state:=888;
		END_IF

 (*запрос на чтение мощности  на всех фазах
--------------------------------------------------------------------------------------------------------------------------------------------------------------------
*)

110:
		tmCheck(in:=FALSE);
		tmCheck(in:=TRUE,pt:=t#2s);
		get_power_done := FALSE;
		get_power(byte1:=16#8, byte2:=16#16, byte3:=16#0,  power_total=>Modbus.pw_total, power1=>Modbus.pw1, power2=>Modbus.pw2,power3=>Modbus.pw3,done=>get_power_done);
		IF get_power_done = TRUE THEN
			state:=111;
		ELSIF tmcheck.Q THEN state:=888;
		END_IF

 (*запрос на чтение энергии T1
--------------------------------------------------------------------------------------------------------------------------------------------------------------------
*)
111:
	tmCheck(in:=FALSE);
		tmCheck(in:=TRUE,pt:=t#2s);
		get_energy_E_T1_done := FALSE;
		get_energy_E_T1(byte1:=5, byte2:=16#0, byte3:=1,  energy=>Modbus.E_T1, done=>get_energy_E_T1_done);
		IF get_energy_E_T1_done = TRUE THEN
			state:=112;
		ELSIF tmcheck.Q THEN state:=888;
		END_IF
 (*запрос на чтение энергии T2
--------------------------------------------------------------------------------------------------------------------------------------------------------------------
*)

112:
	tmCheck(in:=FALSE);
		tmCheck(in:=TRUE,pt:=t#2s);
		get_energy_E_T2_done := FALSE;
		get_energy_E_T2(byte1:=5, byte2:=16#0, byte3:=2,  energy=>Modbus.E_T2, done=>get_energy_E_T2_done);
		IF get_energy_E_T2_done = TRUE THEN
			state:=113;
		ELSIF tmcheck.Q THEN state:=888;
		END_IF


113:
		Timer_day(IN:=NOT Timer_dayQ , PT:=T#10m , Q=>Timer_dayQ , ET=> );
			IF timer_day.q THEN
				state:=114;
			ELSE
				state:=888;
			END_IF

114:
		tmCheck(in:=FALSE);
		tmCheck(in:=TRUE,pt:=t#2s);
		get_energy_MT_done := FALSE;
		get_energy_MT(byte1:=5, byte2:=16#30+INT_TO_BYTE(m), byte3:=INT_TO_BYTE(t),   energy=>energyMT[m,t],done=>get_energy_MT_done);
		IF get_energy_MT_done = TRUE THEN
			t:=t+1;
			IF (t>2 AND m<13) THEN
				t:=1;
				m:=m+1;
				state:=114;
			END_IF

			IF (t>2 AND m>12) THEN
				t:=1;
				m:=1;
				Modbus.M1T1:=energyMT[1,1];
				Modbus.M1T2:=energyMT[1,2];
				Modbus.M2T1:=energyMT[1,1];
				Modbus.M2T2:=energyMT[1,2];
				Modbus.M3T1:=energyMT[1,1];
				Modbus.M3T2:=energyMT[1,2];
				Modbus.M4T1:=energyMT[1,1];
				Modbus.M4T2:=energyMT[1,2];
				Modbus.M5T1:=energyMT[1,1];
				Modbus.M5T2:=energyMT[1,2];
				Modbus.M6T1:=energyMT[1,1];
				Modbus.M6T2:=energyMT[1,2];
				Modbus.M7T1:=energyMT[1,1];
				Modbus.M7T2:=energyMT[1,2];
				Modbus.M8T1:=energyMT[1,1];
				Modbus.M8T2:=energyMT[1,2];
				Modbus.M9T1:=energyMT[1,1];
				Modbus.M9T2:=energyMT[1,2];
				Modbus.M10T1:=energyMT[1,1];
				Modbus.M10T2:=energyMT[1,2];
				Modbus.M11T1:=energyMT[1,1];
				Modbus.M11T2:=energyMT[1,2];
				Modbus.M12T1:=energyMT[1,1];
				Modbus.M12T2:=energyMT[1,2];
				state:=115;
			END_IF
		ELSIF tmcheck.Q THEN state:=888;
		END_IF

888:
		Timer1(IN:=NOT Timer1Q , PT:=tTimerValue , Q=>Timer1Q , ET=> );
		IF timer1.q THEN
			state:=0;
		END_IF

END_CASE

FtrigBusy(CLK:=mb.BUSY );
IF FtrigBusy.Q THEN
	IF mb.Error THEN
		LastModbusError := mb.ErrorDiagnostics;
		LastErrorstate := state;
		CounterError := CounterError + 1;
	ELSE
		CounterSuccess := CounterSuccess + 1;
	END_IF
END_IF



SerialLinecontrolCom1(
	mode:=SerialLinemode_kl6_22b_standard,
	pComIn:=ADR(RS485read.MB.InData),
	pComOut:=ADR(RS485read.MB.OutData),
	SizeComIn:=SIZEOF(RS485read.MB.OutData),
	TxBuffer:=TxBufferCom1,
	RxBuffer:=RxBufferCom1,
	Error=>,
	errorid=>);
END_PROGRAM

(* POU FB_GET_CO2_MH_Z19B, ST *)
FUNCTION_BLOCK FB_GET_CO2_MH_Z19B
VAR_INPUT

END_VAR

VAR_OUTPUT
	co2				: REAL;
	done			: BOOL;
END_VAR

VAR
	SendBuffer		: ARRAY[0..8] OF BYTE;
	ReceiveBuffer	: ARRAY[0..13] OF BYTE;
	Clear			: ClearComBuffer;
	state			: INT:= 0;
	tmcheck			: TON;
	w_CO2		:	WORD;
END_VAR
tmcheck();

CASE state OF

0:
	done:=FALSE;
	Clear(Buffer := RxBufferCom1);
	SendBuffer[0] := 16#FF;
	SendBuffer[1] := 16#01; (* Address *)
	SendBuffer[2] := 16#86;
	SendBuffer[3] := 16#00;
	SendBuffer[4] := 16#00;
	SendBuffer[5] := 16#00;
	SendBuffer[6] := 16#00;
	SendBuffer[7] := 16#00;	(* Checksum *)
	SendBuffer[8] := 16#79;	(* Checksum *)

	SendDataCom1(pSendData:=ADR(SendBuffer),length:=9,TXbuffer:=TXBufferCom1,Busy=>,Error=>);

	tmCheck(in:=FALSE);
	tmCheck(in:=TRUE,pt:=t#2s);
	state:=1;

1: (*ответ*)

	ReceiveDataCom1(pPrefix:=,LenPrefix:=,pSuffix:=,LenSuffix:=,pReceiveData:=ADR(ReceiveBuffer),SizeReceiveData:=9,TImeOut:=t#1s,Reset:=,RXbuffer:=RxBufferCom1,DataReceived=>,busy=>,RxTimeout=>,LenReceiveData=>);

	IF ReceiveDataCom1.Error <> 0 THEN
		state:=9;
	END_IF

	IF ReceiveDataCom1.DataReceived THEN
		state:=2;
	ELSIF tmcheck.Q THEN
		 state:=9;
	END_IF;



2:(*расшифровка*)
	IF (ReceiveBuffer [0] = 16#FF AND ReceiveBuffer [1] = 16#86 ) THEN
		Sensor_CO2_high := ReceiveBuffer [2];
		Sensor_CO2_low := ReceiveBuffer [3];
		MEMCPY(ADR(w_CO2),ADR(ReceiveBuffer[3]),1);
		MEMCPY(ADR(w_CO2)+1,ADR(ReceiveBuffer[2]),1);
		IF (WORD_TO_REAL(w_CO2)<>0 AND WORD_TO_REAL(w_CO2)<5001) THEN
			co2 := WORD_TO_REAL(w_CO2);
			state:=10;
		ELSE
			state:=9;
		END_IF
	ELSE
		state:=9;
	END_IF

9:
	co2:=0;
	done := TRUE;
	state:=0;
10:
	done := TRUE;
	state:=0;

END_CASE;
END_FUNCTION_BLOCK

(* POU FB_GET_SUPPLY, ST *)
FUNCTION_BLOCK FB_GET_SUPPLY
VAR_INPUT
	byte1			: BYTE;
	byte2			: BYTE;
	byte3			: BYTE;

END_VAR

VAR_OUTPUT
	supply1			: REAL;
	supply2			: REAL;
	supply3			: REAL;
	done			: BOOL;
END_VAR

VAR

	Clear			: ClearComBuffer;
	crctest			: WORD;
	arrReceive		: ARRAY[1..12] OF BYTE := 0,0,0,0,0,0,0,0,0,0,0,0;
	arrSend			: ARRAY[1..6] OF BYTE:= 0,0,0,0,0,0;
	state			: INT:= 0;
	dw_DATA		: DWORD:=0;
	tmcheck			: TON;
	CRC_calc		: WORD:=0;
	CRC_get			: WORD:=1;

END_VAR
tmcheck();

CASE state OF

0:

	done:=FALSE;
	Clear(Buffer := RxBufferCom1);

	arrSend[1]:=Merc_address;
	arrSend[2]:=byte1;
	arrSend[3]:=byte2;
	arrSend[4]:=byte3;

	crctest:=F_CRC16(ADR(arrSend), 4);
	MEMCPY(ADR(arrSend)+4,ADR(crctest),2);

	SendDataCom1(pSendData:=ADR(arrSend),length:=6,TXbuffer:=TXBufferCom1 );

	tmCheck(in:=FALSE);
	tmCheck(in:=TRUE,pt:=t#2s);
	state:=1;

1: (*ответ*)

	ReceiveDataCom1(pReceiveData:=ADR(arrReceive),SizeReceiveData:=12,TImeOut:=t#2s,Reset:=,RXbuffer:=RxBufferCom1);

	IF ReceiveDataCom1.Error <> 0 THEN
		state:=9;
	END_IF

	IF ReceiveDataCom1.DataReceived THEN
		state:=2;

	ELSIF tmcheck.Q THEN state:=9;
	END_IF;


2:(*расшифровка*)
	(* arrReceive:=EchoDel(CheckUp:=TRUE, SentA:=arrSend, RecA:=arrReceive, Length:=UDINT_TO_INT(SendDataCom1.Length)); *)
	CRC_calc := F_CRC16(ADR(arrReceive), 10);
	MEMCPY(ADR(CRC_get),ADR(arrReceive[11]),1);
	MEMCPY(ADR(CRC_get)+1,ADR(arrReceive[12]),1);


	IF (  arrReceive[1] = Merc_address  AND CRC_calc = CRC_get ) THEN
		MEMCPY(ADR(dw_DATA),ADR(arrReceive[3]),1);
			MEMCPY(ADR(dw_DATA)+1,ADR(arrReceive[4]),1);
			arrReceive[2]:=arrReceive[2] AND 16#3F;
			MEMCPY(ADR(dw_DATA)+2,ADR(arrReceive[2]),1);
		supply1:=DWORD_TO_REAL(dw_DATA)/100;  (*Вольт*)

		MEMCPY(ADR(dw_DATA),ADR(arrReceive[6]),1);
			MEMCPY(ADR(dw_DATA)+1,ADR(arrReceive[7]),1);
			arrReceive[5]:=arrReceive[5] AND 16#3F;
			MEMCPY(ADR(dw_DATA)+2,ADR(arrReceive[5]),1);
		supply2:=DWORD_TO_REAL(dw_DATA)/100;  (*Вольт*)

		MEMCPY(ADR(dw_DATA),ADR(arrReceive[9]),1);
			MEMCPY(ADR(dw_DATA)+1,ADR(arrReceive[10]),1);
			arrReceive[8]:=arrReceive[8] AND 16#3F;
			MEMCPY(ADR(dw_DATA)+2,ADR(arrReceive[8]),1);
		supply3:=DWORD_TO_REAL(dw_DATA)/100;  (*Вольт*)



			state:=10;
		ELSE state:=9;
	END_IF;

9:
	supply1:=0;
	supply2:=0;
	supply3:=0;
	done := TRUE;
	state:=0;

10:
	done := TRUE;
	state:=0;

END_CASE;
END_FUNCTION_BLOCK

(* POU MB_func/F_CRC16, ST *)
FUNCTION F_CRC16 : WORD
VAR_INPUT
	pData: POINTER TO BYTE;		(* указатель на блок данных *)
	Size: WORD;						(* размер блока  данных *)
END_VAR
VAR
	Cnt: BYTE;							(* счетчик битов *)
END_VAR
F_CRC16 := 16#FFFF;
WHILE Size > 0 DO
	F_CRC16 := F_CRC16 XOR pData^;
	FOR Cnt := 0 TO 7 DO
		IF F_CRC16.0 = 0 THEN
			F_CRC16 := SHR(F_CRC16, 1);
		ELSE
			F_CRC16 := SHR(F_CRC16, 1) XOR 16#A001;
		END_IF
	END_FOR;
	pData := pData + 1;
	Size := Size - 1;
END_WHILE
END_FUNCTION

(* POU FB_GET_CURRENT, ST *)
FUNCTION_BLOCK FB_GET_CURRENT
VAR_INPUT
	byte1			: BYTE;
	byte2			: BYTE;
	byte3			: BYTE;

END_VAR

VAR_OUTPUT
	current1			: REAL;
	current2			: REAL;
	current3			: REAL;
	done			: BOOL;
END_VAR

VAR
	Clear			: ClearComBuffer;
	crctest			: WORD;
	arrReceive		: ARRAY[1..12] OF BYTE := 0,0,0,0,0,0,0,0,0,0,0,0;
	arrSend			: ARRAY[1..6] OF BYTE:= 0,0,0,0,0,0;
	state			: INT:= 0;
	dw_DATA		: DWORD:=0;
	tmcheck			: TON;
	CRC_calc		: WORD:=0;
	CRC_get			: WORD:=1;
END_VAR
tmcheck();

CASE state OF

0:
	done:=FALSE;
	Clear(Buffer := RxBufferCom1);
	arrSend[1]:=Merc_address;
	arrSend[2]:=byte1;
	arrSend[3]:=byte2;
	arrSend[4]:=byte3;

	crctest:=F_CRC16(ADR(arrSend), 4);
	MEMCPY(ADR(arrSend)+4,ADR(crctest),2);

	SendDataCom1(pSendData:=ADR(arrSend),length:=6,TXbuffer:=TXBufferCom1 );

	tmCheck(in:=FALSE);
	tmCheck(in:=TRUE,pt:=t#2s);
	state:=1;

1: (*ответ*)

	ReceiveDataCom1(pReceiveData:=ADR(arrReceive),SizeReceiveData:=12,TImeOut:=t#2s,Reset:=,RXbuffer:=RxBufferCom1);

	IF ReceiveDataCom1.Error <> 0 THEN
		state:=9;
	END_IF

	IF ReceiveDataCom1.DataReceived THEN
		state:=2;
	ELSIF tmcheck.Q THEN state:=9;
	END_IF;


2:(*расшифровка*)

	CRC_calc := F_CRC16(ADR(arrReceive), 10);
	MEMCPY(ADR(CRC_get),ADR(arrReceive[11]),1);
	MEMCPY(ADR(CRC_get)+1,ADR(arrReceive[12]),1);


	IF (  arrReceive[1] = Merc_address  AND CRC_calc = CRC_get ) THEN

			MEMCPY(ADR(dw_DATA),ADR(arrReceive[3]),1);
			MEMCPY(ADR(dw_DATA)+1,ADR(arrReceive[4]),1);
			arrReceive[2]:=arrReceive[2] AND 16#3F;
			MEMCPY(ADR(dw_DATA)+2,ADR(arrReceive[2]),1);
			current1 :=DWORD_TO_REAL(dw_DATA)/1000;  (*Ампер*)

			MEMCPY(ADR(dw_DATA),ADR(arrReceive[6]),1);
			MEMCPY(ADR(dw_DATA)+1,ADR(arrReceive[7]),1);
			arrReceive[5]:=arrReceive[5] AND 16#3F;
			MEMCPY(ADR(dw_DATA)+2,ADR(arrReceive[5]),1);
			current2:=DWORD_TO_REAL(dw_DATA)/1000;  (*Ампер*)

			MEMCPY(ADR(dw_DATA),ADR(arrReceive[9]),1);
			MEMCPY(ADR(dw_DATA)+1,ADR(arrReceive[10]),1);
			arrReceive[8]:=arrReceive[8] AND 16#3F;
			MEMCPY(ADR(dw_DATA)+2,ADR(arrReceive[8]),1);
			current3 :=DWORD_TO_REAL(dw_DATA)/1000;  (*Ампер*)
			state:=10;
		ELSE state:=9;
	END_IF;

9:
	current1:=0;
	current2:=0;
	current3:=0;
	done := TRUE;
	state:=0;
10:
	done := TRUE;
	state:=0;

END_CASE;
END_FUNCTION_BLOCK

(* POU FB_GET_POWER, ST *)
FUNCTION_BLOCK FB_GET_POWER
VAR_INPUT
	byte1			: BYTE;
	byte2			: BYTE;
	byte3			: BYTE;
END_VAR

VAR_OUTPUT
	power_total		: REAL;
	power1			: REAL;
	power2			: REAL;
	power3			: REAL;
	done			: BOOL;
END_VAR

VAR
	Clear				: ClearComBuffer;
	crctest				: WORD;
	arrReceive			: ARRAY[1..15] OF BYTE := 0,0,0,0,0,0,0,0,0,0,0,0,0,0,0;
	arrSend				: ARRAY[1..6] OF BYTE:= 0,0,0,0,0,0;
	state				: INT:= 0;
	dw_DATA			: DWORD:=0;
	tmcheck				: TON;
	CRC_calc			: WORD:=0;
	CRC_get				: WORD:=1;
END_VAR
tmcheck();

CASE state OF

0:
	done:=FALSE;
	Clear(Buffer := RxBufferCom1);
	arrSend[1]:=Merc_address;
	arrSend[2]:=byte1;
	arrSend[3]:=byte2;
	arrSend[4]:=byte3;

	crctest:=F_CRC16(ADR(arrSend), 4);
	MEMCPY(ADR(arrSend)+4,ADR(crctest),2);

	SendDataCom1(pSendData:=ADR(arrSend),length:=6,TXbuffer:=TXBufferCom1 );

	tmCheck(in:=FALSE);
	tmCheck(in:=TRUE,pt:=t#2s);
	state:=1;

1: (*ответ*)

	ReceiveDataCom1(pReceiveData:=ADR(arrReceive),SizeReceiveData:=15,TImeOut:=t#2s,Reset:=,RXbuffer:=RxBufferCom1);

	IF ReceiveDataCom1.Error <> 0 THEN
		state:=9;
	END_IF

	IF ReceiveDataCom1.DataReceived THEN
		state:=2;
	ELSIF tmcheck.Q THEN state:=9;
	END_IF;


2:(*расшифровка*)
	CRC_calc := F_CRC16(ADR(arrReceive), 13);
	MEMCPY(ADR(CRC_get),ADR(arrReceive[14]),1);
	MEMCPY(ADR(CRC_get)+1,ADR(arrReceive[15]),1);


	IF (  arrReceive[1] = Merc_address  AND CRC_calc = CRC_get ) THEN
			MEMCPY(ADR(dw_DATA),ADR(arrReceive[3]),1);
			MEMCPY(ADR(dw_DATA)+1,ADR(arrReceive[4]),1);
			arrReceive[2]:=arrReceive[2] AND 16#3F;
			MEMCPY(ADR(dw_DATA)+2,ADR(arrReceive[2]),1);
			power_total:=DWORD_TO_REAL(dw_DATA)/100;

			MEMCPY(ADR(dw_DATA),ADR(arrReceive[6]),1);
			MEMCPY(ADR(dw_DATA)+1,ADR(arrReceive[7]),1);
			arrReceive[5]:=arrReceive[5] AND 16#3F;
			MEMCPY(ADR(dw_DATA)+2,ADR(arrReceive[5]),1);
			power1:=DWORD_TO_REAL(dw_DATA)/100;

			MEMCPY(ADR(dw_DATA),ADR(arrReceive[9]),1);
			MEMCPY(ADR(dw_DATA)+1,ADR(arrReceive[10]),1);
			arrReceive[8]:=arrReceive[8] AND 16#3F;
			MEMCPY(ADR(dw_DATA)+2,ADR(arrReceive[8]),1);
			power2:=DWORD_TO_REAL(dw_DATA)/100;

			MEMCPY(ADR(dw_DATA),ADR(arrReceive[12]),1);
			MEMCPY(ADR(dw_DATA)+1,ADR(arrReceive[13]),1);
			arrReceive[11]:=arrReceive[11] AND 16#3F;
			MEMCPY(ADR(dw_DATA)+2,ADR(arrReceive[11]),1);
			power3:=DWORD_TO_REAL(dw_DATA)/100;



			state:=10;
		ELSE state:=9;
	END_IF;

9:
	power_total:=0;
	power1:=0;
	power2:=0;
	power3:=0;

	done := TRUE;
	state:=0;
10:
	done := TRUE;
	state:=0;

END_CASE;
END_FUNCTION_BLOCK

(* POU FB_GET_ENERGY, ST *)
FUNCTION_BLOCK FB_GET_ENERGY
VAR_INPUT
	byte1			: BYTE;
	byte2			: BYTE;
	byte3			: BYTE;
END_VAR

VAR_OUTPUT
	energy			: REAL;
	done			: BOOL;
END_VAR

VAR

	Clear				: ClearComBuffer;
	crctest				: WORD;
	arrReceive			: ARRAY[1..22] OF BYTE := 0,0,0,0,0,0,0,0,0,0,0,0,0,0,0,0,0,0,0,0,0,0;
	arrSend				: ARRAY[1..22] OF BYTE:= 0,0,0,0,0,0,0,0,0,0,0,0,0,0,0,0,0,0,0,0,0,0;
	state				: INT:= 0;
	dw_DATA			: DWORD:=0;
	E_active				: REAL:=0;
	E_reactive			: REAL:=0;
	tmcheck				: TON;
	CRC_calc			: WORD:=0;
	CRC_get				: WORD:=1;
END_VAR
tmcheck();

CASE state OF

0:
	done:=FALSE;
	Clear(Buffer := RxBufferCom1);
	arrSend[1]:=Merc_address;
	arrSend[2]:=byte1;
	arrSend[3]:=byte2;
	arrSend[4]:=byte3;

	crctest:=F_CRC16(ADR(arrSend), 4);
	MEMCPY(ADR(arrSend)+4,ADR(crctest),2);

	SendDataCom1(pSendData:=ADR(arrSend),length:=6,TXbuffer:=TXBufferCom1 );

	tmCheck(in:=FALSE);
	tmCheck(in:=TRUE,pt:=t#2s);
	state:=1;

1: (*ответ*)

	ReceiveDataCom1(pReceiveData:=ADR(arrReceive),SizeReceiveData:=19,TImeOut:=t#2s,Reset:=,RXbuffer:=RxBufferCom1);

	IF ReceiveDataCom1.Error <> 0 THEN
		state:=9;
	END_IF

	IF ReceiveDataCom1.DataReceived THEN
		state:=2;
	ELSIF tmcheck.Q THEN state:=9;
	END_IF;


2:(*расшифровка*)
	CRC_calc := F_CRC16(ADR(arrReceive), 17);
	MEMCPY(ADR(CRC_get),ADR(arrReceive[18]),1);
	MEMCPY(ADR(CRC_get)+1,ADR(arrReceive[19]),1);

	IF (  arrReceive[1] = Merc_address  AND CRC_calc = CRC_get ) THEN
			MEMCPY(ADR(dw_DATA),ADR(arrReceive[4]),2);
			MEMCPY(ADR(dw_DATA)+2,ADR(arrReceive[2]),2);
			E_active:=DWORD_TO_REAL(dw_DATA)/1000;(*активная мощ*)
			MEMCPY(ADR(dw_DATA),ADR(arrReceive[12]),2);
			MEMCPY(ADR(dw_DATA)+2,ADR(arrReceive[10]),2);
			E_reactive:=DWORD_TO_REAL(dw_DATA)/1000; (*реактивная мощность*)
			energy:=E_active;
			state:=10;
		ELSE state:=9;
	END_IF;
9:
	energy:=0;
	done := TRUE;
	state:=0;
10:
	done := TRUE;
	state:=0;

END_CASE;
END_FUNCTION_BLOCK

(* POU Thermocontrol, ST *)
PROGRAM Thermocontrol
VAR
(*	period_sec		: INT:=120;  *)  (* Частота работы термостата, секунды*)
	gisterezis		: REAL:=0.2; (*Гистерезис термостата, градусы цельсия *)
	Timer1			: TON;
	Timer1Q			: BOOL;
	state			: INT:=0;
	 tTimerValue		: TIME:=t#120s;  (* Частота работы термостата, секунды*)
END_VAR
(* tTimerValue := DINT_TO_TIME(period_sec*1000); *)

CASE state OF
0:
	IF (Modbus.First_floor_temp > Modbus.First_floor_temp_target+gisterezis ) THEN
		HW_heat_first_floor:=FALSE;
	END_IF

	IF ((Modbus.First_floor_temp <  Modbus.First_floor_temp_target-gisterezis) AND (Modbus.First_floor_temp <>0)  ) THEN
		HW_heat_first_floor:=TRUE;
	END_IF

	state:=1;

1:
	IF (Modbus.Second_floor_temp > Modbus.Second_floor_temp_target+gisterezis ) THEN
		HW_heat_Second_floor:=FALSE;
	END_IF

	IF ((Modbus.Second_floor_temp <  Modbus.Second_floor_temp_target-gisterezis ) AND (Modbus.Second_floor_temp <>0)) THEN
		HW_heat_Second_floor:=TRUE;
	END_IF

	state:=2;
2:
	IF (Modbus.Sport_temp > Modbus.Sport_temp_target+gisterezis ) THEN
		HW_heat_sport:=FALSE;
	END_IF

	IF ((Modbus.Sport_temp <  Modbus.Sport_temp_target-gisterezis ) AND (Modbus.Sport_temp <>0)) THEN
		HW_heat_sport:=TRUE;
	END_IF

	state:=3;

3:
	IF (Modbus.Sauna_temp > Modbus.Sauna_temp_target+gisterezis ) THEN
		HW_heat_Sauna:=FALSE;
	END_IF

	IF ((Modbus.Sauna_temp <  Modbus.Sauna_temp_target-gisterezis ) AND (Modbus.Sauna_temp <>0)) THEN
		HW_heat_Sauna:=TRUE;
	END_IF

	state:=4;

4:
	IF (Modbus.Underfloor_temp > Modbus.Underfloor_temp_target+gisterezis AND Modbus.Underfloor_hum < Modbus.Underfloor_humidity_target-1 ) THEN
		HW_heat_underfloor:=FALSE;
	END_IF

	IF ((Modbus.Underfloor_temp <  Modbus.Underfloor_temp_target-gisterezis OR Modbus.Underfloor_hum > Modbus.Underfloor_humidity_target+1) AND (Modbus.Underfloor_temp <>0)) THEN
		HW_heat_Underfloor:=TRUE;
	END_IF

	state:=100;



100:


	Timer1(IN:=NOT Timer1Q , PT:=tTimerValue , Q=>Timer1Q , ET=> );
		IF timer1.q THEN

		state:=0;
		END_IF



END_CASE
END_PROGRAM

(* POU VentControl, ST *)
PROGRAM VentControl
VAR
	Temperature_max_to_heat	: REAL:=17;		(* Максимальная температура наружнего воздуха при которой разрешено включать воздухонагреватель*)
	gisterezis				: REAL:=0.2;	(* Гистерезис  разрешения включения воздухонагревателя, градусы цельсия *)
	vent_valve_opened	 	: BOOL:=FALSE;	(*После перезагрузки ПЛК считаем что приточный клапан закрыт *)
	Period_start_delay		: INT:=60; 	(* Время задержки включения вентилятора после сигнала на открытие приточного клапана, сек *)
	Period_stop_delay		: INT:=60;		(* Время задержки отключения вентилятора после сигнала на останов вентиляции - для остужения разогретых ТЭНов воздухонагревателя, сек *)
	Timer1					: TON;		(* Таймер задержки включения вентилятора после сигнала на открытие приточного клапана *)
	Timer2					: TON;		(* Таймер задержки отключения вентилятора после сигнала на останов вентиляции - для остужения разогретых ТЭНов воздухонагревателя *)
	Timer1Q					: BOOL;
	Timer2Q					: BOOL;
	tTimerValue1				: TIME;
	tTimerValue2				: TIME;
END_VAR
tTimerValue1 := DINT_TO_TIME(Period_start_delay*1000);
tTimerValue2 := DINT_TO_TIME(Period_stop_delay*1000);

IF (Modbus.Vent=FALSE) THEN
	HW_vent_in_heat := FALSE;
	vent_valve_opened := FALSE;
	HW_vent_valve_input:=FALSE;
	Timer2(IN:=NOT Timer2Q , PT:=tTimerValue2 , Q=>Timer2Q , ET=> );
	IF timer2q THEN
		HW_trans_power:=FALSE;
	END_IF


ELSE
	HW_vent_valve_input:=TRUE;
	HW_vent_valve_output:=TRUE;

	IF (vent_valve_opened = FALSE) THEN
		Timer1(IN:=NOT Timer1Q , PT:=tTimerValue1 , Q=>Timer1Q , ET=> );
		IF timer1.q THEN
			vent_valve_opened := TRUE;
		END_IF
	END_IF

	IF (vent_valve_opened=TRUE) THEN
		HW_trans_power:=TRUE;
(*		IF (HW_vent_reay_pressure=TRUE) THEN	*)

			IF (Modbus.Vent_heat=2) THEN
				IF (Modbus.Street_temp < Temperature_max_to_heat-gisterezis) THEN
					HW_vent_in_heat:=TRUE;
					IF (Modbus.Vent_heat_level=TRUE) THEN
						HW_vent_in_heat_level:=TRUE;
					END_IF
				END_IF
				IF (Modbus.Street_temp > Temperature_max_to_heat+gisterezis) THEN
					HW_vent_in_heat:=FALSE;
				END_IF
			ELSE
				IF (Modbus.Vent_heat=1) THEN
					HW_vent_in_heat:=TRUE;
					IF (Modbus.Vent_heat_level=TRUE) THEN
						HW_vent_in_heat_level:=TRUE;
					ELSE
						HW_vent_in_heat_level:=FALSE;
					END_IF
				END_IF
				IF (Modbus.Vent_heat=0) THEN
					HW_vent_in_heat:=FALSE;
				END_IF
			END_IF
(*		END_IF   *)(*vent_relay_pressure*)
	END_IF (*vent_valve_opened*)
END_IF (*Vent*)
END_PROGRAM

(* POU VentPower, ST *)
PROGRAM VentPower
VAR
	Vent_power			: REAL:=30;  (* После перезагрузки ПЛК задаём начальную мощность условных 30%  *)
	CO2_old				: REAL:=410; (* После перезагрузки ПЛК задаём принудительно последнее значение CO2 = 410 (абсолютно свежий воздух) *)
	Period_vent_switch	: INT:=180; (* Частота переключения режимов работы вентилятора по показаниям датчиков CO2, секунды*)
	Timer1				: TON;
	Timer1Q				: BOOL;
	count				: INT:=0;
	CO2_max			: REAL;
	tTimerValue			: TIME;

END_VAR
tTimerValue := DINT_TO_TIME(Period_vent_switch*1000);

IF (Modbus.Vent =TRUE  ) THEN

	Timer1(IN:=NOT Timer1Q , PT:=tTimerValue , Q=>Timer1Q , ET=> );

	IF timer1.q THEN
	CO2_max:=MAX (Modbus.First_floor_CO2, Modbus.Second_floor_CO2);

	IF (  (CO2_max >=  CO2_old-10 )  AND ( CO2_max >  INT_TO_REAL(Modbus.Target_CO2)*1.05 ) ) THEN
			Vent_power:=Vent_power+5;
		END_IF
		count:=count+1;

		IF (count = 2)	THEN
			IF (  CO2_max <=  INT_TO_REAL(Modbus.Target_CO2)*0.99) THEN
				Vent_power:=Vent_power-1;
			END_IF
		count:=1;
		END_IF

		IF (Vent_power>80) THEN
			Vent_power:=80;
		END_IF
		IF(Vent_power<20) THEN
			Vent_power:=20;
		END_IF

		IF (Vent_Power > 75 AND Modbus.Street_temp > -10  ) THEN

					Modbus.Vent_input_level:=200;	(*200 м. куб в час при подаче напряжения на вентилятор  220V *)
					HW_vent_in_trans_160_220:=FALSE;
					HW_vent_in_trans_LO_HI:=FALSE;

			ELSIF (Vent_Power>50 AND Modbus.Street_temp > -15) THEN
					Modbus.Vent_input_level:=180; (*200 м. куб в час при подаче напряжения на вентилятор 220V *)
					HW_vent_in_trans_160_220:=FALSE;
					HW_vent_in_trans_LO_HI:=FALSE;

			ELSIF (Vent_Power>35  AND Modbus.Street_temp > -20) THEN

					Modbus.Vent_input_level:=150; (* 150 м. куб в час при подаче напряжения на вентилятор160V *)
					HW_vent_in_trans_160_220:=TRUE;
					HW_vent_in_trans_LO_HI:=FALSE;


			ELSIF (Vent_Power>25 ) THEN

					Modbus.Vent_input_level:=110; (* 110 м. куб в час при подаче напряжения на вентилятор 130V *)
					HW_vent_in_trans_105_130:=FALSE;
					HW_vent_in_trans_LO_HI:=TRUE;


			ELSE
				Modbus.Vent_input_level:=80; (* 80 м. куб в час при подаче напряжения на вентилятор 105V *)
				HW_vent_in_trans_105_130:=TRUE;
				HW_vent_in_trans_LO_HI:=TRUE;


			END_IF

			CO2_old:=CO2_max;

		END_IF	(* Timer1 *)

	ELSE	 (* Vent=TRUE*)


		Modbus.Vent_input_level:=0;

END_IF   (* Vent=TRUE*)
END_PROGRAM

(* POU Poliv, ST *)
PROGRAM Poliv
VAR
	TRIG_poliv_terrasa	:	R_TRIG;
	TRIG_poliv_zapad	:	R_TRIG;
	TRIG_poliv_south		:	R_TRIG;
	TRIG_poliv_north		:	R_TRIG;

	Period_pomp_garden_delay	: INT:=15;				(* Задержка включения насоса после сигнала на открытие клапана=15 сек. *)

 	 tTimerValue_zapad			: TIME;
	Timer_poliv_zapad			: TON;
	Timer_poliv_zapadQ			:  BOOL;
	 tTimerValue_zapad_est		: TIME;

	tTimerValue_terrasa			: TIME;
	Timer_poliv_terrasa			: TON;
	Timer_poliv_terrasaQ			:  BOOL;
	tTimerValue_terrasa_est		: TIME;

	 tTimerValue_south			: TIME;
	Timer_poliv_south				: TON;
	Timer_poliv_southQ			:  BOOL;
	 tTimerValue_south_est		: TIME;


 	tTimerValue_north				: TIME;
	Timer_poliv_north				: TON;
	Timer_poliv_northQ			:  BOOL;
 	tTimerValue_north_est			: TIME;

	TON_pomp_garden			: TON ;
	pomp_garden_start			: BOOL;

	tTimerValue					: TIME;
END_VAR
tTimerValue := DINT_TO_TIME(Period_pomp_garden_delay*1000);


Timer_poliv_zapad();
Timer_poliv_terrasa();
Timer_poliv_south();
Timer_poliv_north();

TRIG_poliv_terrasa(CLK :=HW_button_poliv_terrasa);
TRIG_poliv_zapad(CLK :=HW_button_poliv_zapad);
TRIG_poliv_south(CLK :=HW_button_poliv_south);
TRIG_poliv_north(CLK :=HW_button_poliv_north);


IF (TRIG_poliv_terrasa.Q) THEN
	IF (Modbus.Poliv_terrasa = TRUE ) THEN
		Modbus.Poliv_terrasa := FALSE;
		iobroker.Poliv_terrasa := FALSE;
	ELSE
		iobroker.Poliv_terrasa := TRUE;
		Modbus.Poliv_terrasa := TRUE;
		Modbus.Poliv_terrasa_minutes:=120;
	END_IF

END_IF



IF (TRIG_poliv_zapad.Q) THEN
	IF (Modbus.Poliv_zapad = TRUE ) THEN
		iobroker.Poliv_zapad:=FALSE;
		Modbus.Poliv_zapad := FALSE;
	ELSE
		iobroker.Poliv_zapad:=TRUE;
		Modbus.Poliv_zapad := TRUE;
		Modbus.Poliv_zapad_minutes:=120;
	END_IF

END_IF


IF (TRIG_poliv_south.Q) THEN
	IF (Modbus.Poliv_south = TRUE ) THEN
		iobroker.Poliv_south := FALSE;
		Modbus.Poliv_south := FALSE;
	ELSE
		iobroker.Poliv_south := TRUE;
		Modbus.Poliv_south_minutes:=120;
		Modbus.Poliv_south := TRUE;
	END_IF

END_IF


IF (TRIG_poliv_north.Q) THEN
	IF (Modbus.Poliv_north = TRUE ) THEN
		iobroker.Poliv_north := FALSE;
		Modbus.Poliv_north := FALSE;
	ELSE
		iobroker.Poliv_north := TRUE;
		Modbus.Poliv_north_minutes:=120;
		Modbus.Poliv_north := TRUE;
	END_IF

END_IF


Modbus.Poliv_zapad_minutes_est	:= TIME_TO_INT(tTimerValue_zapad_est)/(60*1000);
Modbus.Poliv_terrasa_minutes_est	:=  TIME_TO_INT(tTimerValue_zapad_est)/(60*1000);
Modbus.Poliv_south_minutes_est	:=  TIME_TO_INT(tTimerValue_south_est)/(60*1000);
Modbus.Poliv_north_minutes_est	:=  TIME_TO_INT(tTimerValue_north_est)/(60*1000);


IF (Modbus.Poliv_zapad = TRUE ) THEN
	tTimerValue_zapad := DINT_TO_TIME(Modbus.Poliv_zapad_minutes*60*1000);
	HW_poliv_zapad	:=	TRUE;
	Timer_poliv_zapad(IN:=NOT Timer_poliv_zapadQ , PT:=tTimerValue_zapad , Q=>Timer_poliv_zapadQ , ET=>tTimerValue_zapad_est );

END_IF
IF (Modbus.Poliv_zapad = FALSE ) THEN
	HW_poliv_zapad	:=	FALSE;
	Timer_poliv_zapadQ := FALSE;
	Timer_poliv_zapad(IN:=FALSE , PT:=T#0ms , Q=>Timer_poliv_zapadQ , ET=>tTimerValue_zapad_est );
END_IF
IF Timer_poliv_zapad.q THEN
	Modbus.Poliv_zapad := FALSE;
	HW_poliv_zapad	:=	FALSE;
END_IF




IF (Modbus.Poliv_terrasa = TRUE ) THEN
	tTimerValue_terrasa := DINT_TO_TIME(Modbus.Poliv_terrasa_minutes*60*1000);
	HW_poliv_terrasa	:=	TRUE;
	Timer_poliv_terrasa(IN:=NOT Timer_poliv_terrasaQ , PT:=tTimerValue_terrasa , Q=>Timer_poliv_terrasaQ , ET=>tTimerValue_terrasa_est );
END_IF
IF (Modbus.Poliv_terrasa = FALSE ) THEN
	HW_poliv_terrasa	:=	FALSE;
	Timer_poliv_terrasaQ := FALSE;
	Timer_poliv_terrasa(IN:=FALSE , PT:=T#0ms , Q=>Timer_poliv_terrasaQ , ET=>tTimerValue_terrasa_est );
END_IF
IF Timer_poliv_terrasa.q THEN
	Modbus.Poliv_terrasa := FALSE;
	HW_poliv_zapad	:=	FALSE;
END_IF



IF (Modbus.Poliv_south = TRUE ) THEN
	tTimerValue_south := DINT_TO_TIME(Modbus.Poliv_south_minutes*60*1000);
	HW_poliv_south	:=	TRUE;
	Timer_poliv_south(IN:=NOT Timer_poliv_southQ , PT:=tTimerValue_south , Q=>Timer_poliv_southQ , ET=>tTimerValue_south_est );
END_IF
IF (Modbus.Poliv_south = FALSE ) THEN
	HW_poliv_south	:=	FALSE;
	Timer_poliv_southQ := FALSE;
	Timer_poliv_south(IN:=FALSE , PT:=T#0ms , Q=>Timer_poliv_southQ , ET=>tTimerValue_south_est );
END_IF
IF Timer_poliv_south.q THEN
	Modbus.Poliv_south := FALSE;
	HW_poliv_south	:=	FALSE;
END_IF



IF (Modbus.Poliv_north = TRUE ) THEN
	tTimerValue_north := DINT_TO_TIME(Modbus.Poliv_north_minutes*60*1000);
	HW_poliv_north	:=	TRUE;
	Timer_poliv_north(IN:=NOT Timer_poliv_northQ , PT:=tTimerValue_north , Q=>Timer_poliv_northQ , ET=>tTimerValue_north_est );
END_IF
IF (Modbus.Poliv_north = FALSE ) THEN
	HW_poliv_north	:=	FALSE;
	Timer_poliv_northQ := FALSE;
	Timer_poliv_north(IN:=FALSE , PT:=T#0ms , Q=>Timer_poliv_northQ , ET=>tTimerValue_north_est );
END_IF
IF Timer_poliv_north.q THEN
	Modbus.Poliv_north := FALSE;
	HW_poliv_north	:=	FALSE;
END_IF






IF ((HW_poliv_zapad=TRUE OR HW_poliv_terrasa=TRUE 	OR HW_poliv_south =	TRUE OR HW_poliv_north = TRUE) AND (HW_pomp_Garden=FALSE)  )  THEN
	pomp_garden_start			:=TRUE;
END_IF


TON_pomp_garden(IN := pomp_garden_start, PT:= tTimerValue);
Modbus.Pomp_garden	 	:= TON_pomp_garden.Q;
HW_Pomp_garden		:= TON_pomp_garden.Q;

IF (HW_poliv_zapad=FALSE AND HW_poliv_terrasa=FALSE 	AND HW_poliv_south = FALSE  AND HW_poliv_north = FALSE)   THEN
	pomp_garden_start		:= FALSE;
	Modbus.Pomp_garden	 	:= FALSE;
	HW_Pomp_garden		:= FALSE;
END_IF
END_PROGRAM

(* POU Power_act, ST *)
PROGRAM Power_act
VAR
	fbCalcSunriseSunset   	: FB_CalcSunriseSunset;
	todSunrise            		: TOD;
   	todSunset          		: TOD;
	dtCurrentDate         		: DT;
	fileTime              		: T_FILETIME;
	fbGetSystemTime       	: GETSYSTEMTIME;
	time_now			: TOD;
	tz					: TIME:=T#5h;


END_VAR
fbGetSystemTime(timeLoDW =>fileTime.dwLowDateTime,
                timeHiDW =>fileTime.dwHighDateTime);
dtCurrentDate:=FILETIME_TO_DT(fileTime);


fbCalcSunriseSunset( fDegreeOfLongitude := 73.26,   (* Longitude of Verl *)
                     fDegreeOfLatitude := 61.15,   (* Latitude of Verl *)
                     fReferenceMeridian := 73.26,  (* Central European Summer Time *)
                     dCurrentDate := DT_TO_DATE(dtCurrentDate),
                     todSunrise => todSunrise,
                     todSunset => todSunset);

time_now	:= DT_TO_TOD(dtCurrentDate)+tz;

IF ( time_now > todSunrise  AND  time_now < todSunset   ) THEN
		Modbus.Light_reserv := FALSE;
	ELSE
		IF (Modbus.Security_status = FALSE) THEN
			Modbus.Light_reserv := TRUE;
		END_IF
END_IF

IF (Modbus.Security_status = TRUE) THEN
	Modbus.Light_reserv := FALSE;
END_IF



IF (Modbus.Light_reserv=TRUE AND (Modbus.Light_reserv_manual=1 OR Modbus.Light_reserv_manual=2)) THEN
		HW_light_rezerv:=TRUE;
	ELSIF  (Modbus.Light_reserv=TRUE AND  Modbus.Light_reserv_manual=0 ) THEN
		HW_light_rezerv:=FALSE;
	ELSIF (Modbus.Light_reserv=FALSE AND Modbus.Light_reserv_manual=1) THEN
		HW_light_rezerv:=TRUE;
	ELSE
		HW_light_rezerv:=FALSE;
END_IF
END_PROGRAM

(* POU Buttons, ST *)
PROGRAM Buttons
VAR
(*	TRIG_BUT_light1			:	R_TRIG;
	TRIG_BUT_light_kitchen	:	R_TRIG;
	TRIG_BUT_light_terrasa	:	R_TRIG;
*)
	SW_LIGHT_GARDEN			: SM_BUTT;		(* вкл/откл прожектор *)
	SW_VOROTA				: FB_ShortLongClick;
	TRIG_vorota_open			: R_TRIG;
	TRIG_vorota_modbus			: R_TRIG;
	TRIG_vorota_open_modbus	: R_TRIG;
(*	SW_VOROTA				: SM_BUTT; *)

(*	Vorota_switch					: BOOL:=FALSE; *)
	Vorota_open					: BOOL:=FALSE;

	Pulse						: TP;
	PT_length					: TIME:= T#500ms;


	Timer_vo					: TON;
	Timer_voQ					: BOOL;
	tTimerValue_vo				: TIME:= T#23500ms;





END_VAR
	SW_LIGHT_GARDEN		(IN:=HW_button_light_garden, IN1:=Modbus.Light_garden, 	Q=>Modbus.Light_garden);		(* Конпка *)
	SW_VOROTA			(bSwitch :=HW_button_vorota, tSwitchTime   := t#2000ms);

	iobroker.Vorota_active:=FALSE;
	Timer_vo();

	TRIG_vorota_modbus(CLK :=Modbus.Vorota);
	TRIG_vorota_open_modbus(CLK :=Modbus.Vorota_open);

	IF TRIG_vorota_modbus.Q		THEN
		Pulse (IN:=TRUE, PT:=PT_length, Q=>HW_vorota , ET=> );
	END_IF

	Pulse (IN:=SW_VOROTA.bShortClick, PT:=PT_length, Q=>HW_vorota , ET=> );

(*	HW_vorota					:=	Modbus.Vorota; *)

	IF (SW_VOROTA.bShortClick) THEN
		iobroker.Vorota_active:=TRUE;
	END_IF




	IF (SW_VOROTA.bLongClick OR TRIG_vorota_open_modbus.Q) THEN
		Vorota_open				:= TRUE;
		iobroker.Vorota_open_active:=TRUE;
	END_IF

	Pulse (IN:=SW_VOROTA.bLongClick, PT:=PT_length, Q=>HW_vorota , ET=> );
	Pulse (IN:=TRIG_vorota_open_modbus.Q, PT:=PT_length, Q=>HW_vorota , ET=> );

	IF 	Vorota_open		THEN
		Timer_vo(IN:=NOT Timer_voQ , PT:=tTimerValue_vo , Q=>Timer_voQ , ET=> );
	END_IF

	TRIG_vorota_open(CLK :=Timer_voQ);

	IF TRIG_vorota_open.Q		THEN
		Pulse (IN:=TRUE, PT:=PT_length, Q=>HW_vorota , ET=> );
		Vorota_open				:= FALSE;
		iobroker.Vorota_open_active:=FALSE;
	END_IF
END_PROGRAM

(* POU SM_BUTT, ST *)
FUNCTION_BLOCK SM_BUTT            (* ФУНКЦИОНАЛЬНЫЙ БЛОК ДЛЯ ПРОСТОЙ КНОПКИ *)
    VAR_INPUT
       	IN: BOOL;          	(*ВХОД ЗА КОТОРЫМ МЫ СЛЕДИМ *)
	IN1:BOOL;				(*ВЫХОД ЗА КОТОРЫМ ТОЖЕ СЛЕДИМ*)
    END_VAR

    VAR_OUTPUT
	Q : BOOL;        			(*СОСТОЯНИЕ ВЫХОДА*)
    END_VAR
    VAR
  MEM : BOOL;    			(* ВНУТРЕННЯЯ ПЕРЕМЕННАЯ ДЛЯ ХРАНЕНИЯ СОСТОЯНИЯ КНОПКИ *)
    END_VAR
Q:=IN1;

IF IN AND NOT MEM THEN 	(* ПОЙМАЛИ ПЕРЕДНИЙ ФРОНТ - НАЖАЛИ НА КНОПКУ *)
	Q := NOT IN1;    			(* МЕНЯЕМ СОСТОЯНИЕ ВЫХОДА НА ПРОТИВОПОЛОЖНОЕ *)
END_IF

MEM := IN;                       		(* ЗАПОМИНАЕМ ТЕКУЩЕЕ ЗНАЧЕНИЕ КНОПКИ *)
END_FUNCTION_BLOCK

(* POU Mqtt, ST *)
PROGRAM Mqtt
VAR
	FB_Mqtt_Controller 		: FB_Mqtt_Controller_V10;
	stMqttSettings				: ST_MqttSettings;
	bMqttControllerBusy		: BOOL;

	FB_Mqtt_Publish1 			: FB_Mqtt_Publish_V10;
	FB_Mqtt_Publish2			: FB_Mqtt_Publish_V10;
	FB_Mqtt_Publish3			: FB_Mqtt_Publish_V10;
	FB_Mqtt_Publish4			: FB_Mqtt_Publish_V10;
	FB_Mqtt_Publish5			: FB_Mqtt_Publish_V10;
	FB_Mqtt_Publish6			: FB_Mqtt_Publish_V10;
	FB_Mqtt_Publish7			: FB_Mqtt_Publish_V10;
	FB_Mqtt_Publish8			: FB_Mqtt_Publish_V10;
	FB_Mqtt_Publish9			: FB_Mqtt_Publish_V10;
	FB_Mqtt_Publish10		: FB_Mqtt_Publish_V10;
	FB_Mqtt_Publish11		: FB_Mqtt_Publish_V10;
	FB_Mqtt_Publish12		: FB_Mqtt_Publish_V10;
	FB_Mqtt_Publish13 		: FB_Mqtt_Publish_V10;
	FB_Mqtt_Publish14		: FB_Mqtt_Publish_V10;
	FB_Mqtt_Publish15		: FB_Mqtt_Publish_V10;
	FB_Mqtt_Publish16		: FB_Mqtt_Publish_V10;
	FB_Mqtt_Publish17		: FB_Mqtt_Publish_V10;
	FB_Mqtt_Publish18		: FB_Mqtt_Publish_V10;
	FB_Mqtt_Publish19		: FB_Mqtt_Publish_V10;
	FB_Mqtt_Publish20		: FB_Mqtt_Publish_V10;
	FB_Mqtt_Publish21		: FB_Mqtt_Publish_V10;
	FB_Mqtt_Publish22		: FB_Mqtt_Publish_V10;
	FB_Mqtt_Publish23		: FB_Mqtt_Publish_V10;
	FB_Mqtt_Publish24		: FB_Mqtt_Publish_V10;
	FB_Mqtt_Publish25		: FB_Mqtt_Publish_V10;
	FB_Mqtt_Publish26		: FB_Mqtt_Publish_V10;
	FB_Mqtt_Publish27		: FB_Mqtt_Publish_V10;
	FB_Mqtt_Publish28		: FB_Mqtt_Publish_V10;

	bPublishBusy1			: BOOL;
	bPublishBusy2			: BOOL;
	bPublishBusy3			: BOOL;
	bPublishBusy4			: BOOL;
	bPublishBusy5			: BOOL;
	bPublishBusy6			: BOOL;
	bPublishBusy7			: BOOL;
	bPublishBusy8			: BOOL;
	bPublishBusy9			: BOOL;
	bPublishBusy10			: BOOL;
	bPublishBusy11			: BOOL;
	bPublishBusy12			: BOOL;
	bPublishBusy13			: BOOL;
	bPublishBusy14			: BOOL;
	bPublishBusy15			: BOOL;
	bPublishBusy16			: BOOL;
	bPublishBusy17			: BOOL;
	bPublishBusy18			: BOOL;
	bPublishBusy19			: BOOL;
	bPublishBusy20			: BOOL;
	bPublishBusy21			: BOOL;
	bPublishBusy22			: BOOL;
	bPublishBusy23			: BOOL;
	bPublishBusy24			: BOOL;
	bPublishBusy25			: BOOL;
	bPublishBusy26			: BOOL;
	bPublishBusy27			: BOOL;
	bPublishBusy28			: BOOL;

	START: BOOL;
END_VAR
FB_Mqtt_Controller (
		bActive			:= TRUE,
		sMqttClientId		:= 'plc',
		sMqttUserId		:= 'mqtt',
		sMqttPassword	:= 'mqtt',
		sMqttBrokerIp		:= '192.168.2.200',
		nMqttBrokerPort	:= 1883,
		stMqttSettings		:= stMqttSettings,
		bBusy			=> bMqttControllerBusy
	);

IF NOT bMqttControllerBusy THEN

	FB_Mqtt_Publish1(sTopic:='BECKHOFF_CX9000/Mercury/M1T1',sValue:=REAL_TO_STRING(Mercury.M1T1),bRetain:=FALSE, stMqttSettings:=stMqttSettings,bBusy => bPublishBusy1 );
	FB_Mqtt_Publish2(sTopic:='BECKHOFF_CX9000/Mercury/M1T2',sValue:=REAL_TO_STRING(Mercury.M1T2),bRetain:=FALSE, stMqttSettings:=stMqttSettings,bBusy => bPublishBusy2 );
	FB_Mqtt_Publish3(sTopic:='BECKHOFF_CX9000/Mercury/M2T1',sValue:=REAL_TO_STRING(Mercury.M2T1),bRetain:=FALSE, stMqttSettings:=stMqttSettings,bBusy => bPublishBusy3 );
	FB_Mqtt_Publish4(sTopic:='BECKHOFF_CX9000/Mercury/M2T2',sValue:=REAL_TO_STRING(Mercury.M2T2),bRetain:=FALSE, stMqttSettings:=stMqttSettings,bBusy => bPublishBusy4 );
	FB_Mqtt_Publish5(sTopic:='BECKHOFF_CX9000/Mercury/M3T1',sValue:=REAL_TO_STRING(Mercury.M3T1),bRetain:=FALSE, stMqttSettings:=stMqttSettings,bBusy => bPublishBusy5 );
	FB_Mqtt_Publish6(sTopic:='BECKHOFF_CX9000/Mercury/M3T2',sValue:=REAL_TO_STRING(Mercury.M3T2),bRetain:=FALSE, stMqttSettings:=stMqttSettings,bBusy => bPublishBusy6 );
	FB_Mqtt_Publish7(sTopic:='BECKHOFF_CX9000/Mercury/M4T1',sValue:=REAL_TO_STRING(Mercury.M4T1),bRetain:=FALSE, stMqttSettings:=stMqttSettings,bBusy => bPublishBusy7 );
	FB_Mqtt_Publish8(sTopic:='BECKHOFF_CX9000/Mercury/M4T2',sValue:=REAL_TO_STRING(Mercury.M4T2),bRetain:=FALSE, stMqttSettings:=stMqttSettings,bBusy => bPublishBusy8 );
	FB_Mqtt_Publish9(sTopic:='BECKHOFF_CX9000/Mercury/M5T1',sValue:=REAL_TO_STRING(Mercury.M5T1),bRetain:=FALSE, stMqttSettings:=stMqttSettings,bBusy => bPublishBusy9 );
	FB_Mqtt_Publish10(sTopic:='BECKHOFF_CX9000/Mercury/M5T2',sValue:=REAL_TO_STRING(Mercury.M5T2),bRetain:=FALSE, stMqttSettings:=stMqttSettings,bBusy => bPublishBusy10 );
	FB_Mqtt_Publish11(sTopic:='BECKHOFF_CX9000/Mercury/M6T1',sValue:=REAL_TO_STRING(Mercury.M6T1),bRetain:=FALSE, stMqttSettings:=stMqttSettings,bBusy => bPublishBusy11 );
	FB_Mqtt_Publish12(sTopic:='BECKHOFF_CX9000/Mercury/M6T2',sValue:=REAL_TO_STRING(Mercury.M6T2),bRetain:=FALSE, stMqttSettings:=stMqttSettings,bBusy => bPublishBusy12 );
	FB_Mqtt_Publish13(sTopic:='BECKHOFF_CX9000/Mercury/M7T1',sValue:=REAL_TO_STRING(Mercury.M7T1),bRetain:=FALSE, stMqttSettings:=stMqttSettings,bBusy => bPublishBusy13 );
	FB_Mqtt_Publish14(sTopic:='BECKHOFF_CX9000/Mercury/M7T2',sValue:=REAL_TO_STRING(Mercury.M7T2),bRetain:=FALSE, stMqttSettings:=stMqttSettings,bBusy => bPublishBusy14);
	FB_Mqtt_Publish15(sTopic:='BECKHOFF_CX9000/Mercury/M8T1',sValue:=REAL_TO_STRING(Mercury.M8T1),bRetain:=FALSE, stMqttSettings:=stMqttSettings,bBusy => bPublishBusy15 );
	FB_Mqtt_Publish16(sTopic:='BECKHOFF_CX9000/Mercury/M8T2',sValue:=REAL_TO_STRING(Mercury.M8T2),bRetain:=FALSE, stMqttSettings:=stMqttSettings,bBusy => bPublishBusy16 );
	FB_Mqtt_Publish17(sTopic:='BECKHOFF_CX9000/Mercury/M9T1',sValue:=REAL_TO_STRING(Mercury.M9T1),bRetain:=FALSE, stMqttSettings:=stMqttSettings,bBusy => bPublishBusy17 );
	FB_Mqtt_Publish18(sTopic:='BECKHOFF_CX9000/Mercury/M9T2',sValue:=REAL_TO_STRING(Mercury.M9T2),bRetain:=FALSE, stMqttSettings:=stMqttSettings,bBusy => bPublishBusy18 );
	FB_Mqtt_Publish19(sTopic:='BECKHOFF_CX9000/Mercury/M10T1',sValue:=REAL_TO_STRING(Mercury.M10T1),bRetain:=FALSE, stMqttSettings:=stMqttSettings,bBusy => bPublishBusy19 );
	FB_Mqtt_Publish20(sTopic:='BECKHOFF_CX9000/Mercury/M10T2',sValue:=REAL_TO_STRING(Mercury.M10T2),bRetain:=FALSE, stMqttSettings:=stMqttSettings,bBusy => bPublishBusy20 );
	FB_Mqtt_Publish21(sTopic:='BECKHOFF_CX9000/Mercury/M11T1',sValue:=REAL_TO_STRING(Mercury.M11T1),bRetain:=FALSE, stMqttSettings:=stMqttSettings,bBusy => bPublishBusy21 );
	FB_Mqtt_Publish22(sTopic:='BECKHOFF_CX9000/Mercury/M11T2',sValue:=REAL_TO_STRING(Mercury.M11T2),bRetain:=FALSE, stMqttSettings:=stMqttSettings,bBusy => bPublishBusy22 );
	FB_Mqtt_Publish23(sTopic:='BECKHOFF_CX9000/Mercury/M12T1',sValue:=REAL_TO_STRING(Mercury.M12T1),bRetain:=FALSE, stMqttSettings:=stMqttSettings,bBusy => bPublishBusy23 );
	FB_Mqtt_Publish24(sTopic:='BECKHOFF_CX9000/Mercury/M12T2',sValue:=REAL_TO_STRING(Mercury.M12T2),bRetain:=FALSE, stMqttSettings:=stMqttSettings,bBusy => bPublishBusy24 );
	FB_Mqtt_Publish25(sTopic:='BECKHOFF_CX9000/Sensors/Control_hum',sValue:=REAL_TO_STRING(iob_mqtt.Control_hum),bRetain:=FALSE, stMqttSettings:=stMqttSettings,bBusy => bPublishBusy25 );
	FB_Mqtt_Publish26(sTopic:='BECKHOFF_CX9000/Sensors/Control_temp',sValue:=REAL_TO_STRING(iob_mqtt.Control_temp),bRetain:=FALSE, stMqttSettings:=stMqttSettings,bBusy => bPublishBusy26 );
	FB_Mqtt_Publish27(sTopic:='BECKHOFF_CX9000/Sensors/Control_hum2',sValue:=REAL_TO_STRING(iob_mqtt.Control_hum2),bRetain:=FALSE, stMqttSettings:=stMqttSettings,bBusy => bPublishBusy27 );
	FB_Mqtt_Publish28(sTopic:='BECKHOFF_CX9000/Sensors/Control_temp2',sValue:=REAL_TO_STRING(iob_mqtt.Control_temp2),bRetain:=FALSE, stMqttSettings:=stMqttSettings,bBusy => bPublishBusy28 );

END_IF
(*    END    SEND DATA VIA MQTT  *)
END_PROGRAM

(* POU FB_Mqtt_Controller_V10, ST *)
(* @NESTEDCOMMENTS := 'Yes' *)
(* @PATH := '\/_Generic\/Mqtt' *)
(* @OBJECTFLAGS := '0, 8' *)
(* @SYMFILEFLAGS := '2048' *)
FUNCTION_BLOCK FB_Mqtt_Controller_V10
VAR_INPUT
(*	bActive			: BOOL := FALSE;
	sMqttClientId	: STRING[23]:='plc';
	sMqttUserId	: STRING[25] := 'mqtt';
	sMqttPassword	: STRING[25] := 'mqtt';
	sMqttBrokerIP	: STRING[15]:='192.168.3.200';
	nMqttBrokerPort	: UDINT := 1883;
*)
	bActive			: BOOL := FALSE;
	sMqttClientId	: STRING[23];
	sMqttUserId	: STRING[25] := '';
	sMqttPassword	: STRING[25] := '';
	sMqttBrokerIP	: STRING[15];
	nMqttBrokerPort	: UDINT := 1883;
END_VAR
VAR_OUTPUT
	bBusy	: BOOL := FALSE;
END_VAR
VAR_IN_OUT
	stMqttSettings	: ST_MqttSettings;
END_VAR
VAR
	iState			: INT := 0;
	fbSocketConnect	: FB_SocketConnect;
	fbSocketClose	: FB_SocketClose;

	fbMqttTelegramConnect	: FB_MqttTelegram_Connect_V10;
	fbMqttTelegramPingReq	: FB_MqttTelegram_PingReq_V10;
	fbMqttSend				: FB_Mqtt_Send_V10;
	fbMqttReceive			: FB_Mqtt_Receive_V10;
END_VAR
VAR CONSTANT
	C_STARTUP					: INT := 0;
	C_CONNECT					: INT := 100;
	C_CONNECT_WAIT				: INT := 110;
	C_CLOSE						: INT := 200;
	C_CLOSE_WAIT				: INT := 210;
	C_IDLE						: INT := 500;
END_VAR
(* @END_DECLARATION := '0' *)
(*
 * Connects to mqtt broker
 * Sends connect message
 * Sends ping(back)
 * Sends disconnect
 *)
CASE iState OF
	C_STARTUP:
		stMqttSettings.bConnected			:= FALSE;
		stMqttSettings.bConnectPackageSent	:= FALSE;
		stMqttSettings.bDisconnect			:= FALSE;
		stMqttSettings.bSocketConnection	:= FALSE;
		stMqttSettings.bError				:= FALSE;
		stMqttSettings.bValidConnection		:= FALSE;
		stMqttSettings.wPackageIdentifier	:= 1;
		stMqttSettings.bActive				:= bActive;
		stMqttSettings.hSocket				:= fbSocketConnect.hSocket;
		stMqttSettings.nMqttBrokerPort		:= nMqttBrokerPort;
		stMqttSettings.sMqttBrokerIP		:= sMqttBrokerIP;
		stMqttSettings.sMqttClientId		:= sMqttClientId;
		stMqttSettings.sMqttUserId		:= sMqttUserId;
		stMqttSettings.sMqttPassword		:= sMqttPassword;

		stMqttSettings.stMqttReceivedTelegram.nDataLength := 0;

		bBusy := FALSE;

		CallMqttBlocks();

		IF bActive THEN
			iState := C_CONNECT;
		END_IF;

	(* Start connection *)
	C_CONNECT:
		bBusy := TRUE;

		fbSocketConnect(
			bExecute	:= FALSE
		);

		fbSocketConnect(
			sSrvNetId	:= '',
			sRemoteHost	:= sMqttBrokerIP,
			nRemotePort	:= nMqttBrokerPort,
			bExecute	:= TRUE,
			tTimeout	:= USINT_TO_TIME(stMqttSettings.usKeepAliveTime) + t#10s
		);

		iState := C_CONNECT_WAIT;

	(* Wait till connected *)
	C_CONNECT_WAIT:
		fbSocketConnect(
			bExecute := FALSE
		);

		IF
			NOT fbSocketConnect.bBusy
			AND NOT fbSocketConnect.bError
		THEN
			iState 								:= C_IDLE;
			stMqttSettings.hSocket				:= fbSocketConnect.hSocket;
			stMqttSettings.bSocketConnection	:= TRUE;
		END_IF;

		IF fbSocketConnect.bError THEN
			iState := C_STARTUP;
		END_IF;

		IF NOT stMqttSettings.bActive THEN
			iState := C_STARTUP;
		END_IF;

	(* Close connection *)
	C_CLOSE:
		bBusy := TRUE;

		fbSocketClose(
			bExecute	:= TRUE,
			hSocket		:= stMqttSettings.hSocket
		);

		iState := C_CLOSE_WAIT;

	(* Wait close connection *)
	C_CLOSE_WAIT:
		fbSocketClose(
			bExecute := FALSE
		);

		IF
			NOT fbSocketClose.bBusy
			AND NOT fbSocketClose.bError
		THEN
			iState := C_STARTUP;
		END_IF;

		IF fbSocketClose.bError THEN
			iState := C_STARTUP;
		END_IF;

		IF NOT stMqttSettings.bActive THEN
			iState := C_STARTUP;
		END_IF;

	(* Idle *)
	C_IDLE:
		bBusy 					:= FALSE;
		stMqttSettings.bActive	:= bActive;

		stMqttSettings.bValidConnection :=
			NOT stMqttSettings.bError
			AND NOT stMqttSettings.bDisconnect
			AND stMqttSettings.bConnected
			AND stMqttSettings.bSocketConnection
			AND stMqttSettings.bActive;

		CallMqttBlocks();

		IF
			stMqttSettings.bDisconnect
			OR stMqttSettings.bError
			OR NOT stMqttSettings.bActive
		THEN
			IF
				stMqttSettings.bConnected
				OR stMqttSettings.bSocketConnection
			THEN
				(* TODO : send disconnect *)
				iState := C_CLOSE;
			ELSE
				iState := C_CLOSE;
			END_IF;
		END_IF;

	ELSE
		iState := C_STARTUP;
END_CASE;
(*	END_FUNCTION_BLOCK	*)
END_FUNCTION_BLOCK
ACTION CallMqttBlocks:
(*ACTION	CallMqttBlocks: *)
fbMqttReceive(
	stMqttSettings := stMqttSettings
);

fbMqttTelegramConnect(
	stMqttSettings := stMqttSettings
);

fbMqttTelegramPingReq(
	stMqttSettings := stMqttSettings
);

fbMqttSend(
	stMqttSettings := stMqttSettings
);

(* END_ACTION *)
END_ACTION

(* POU Intern/FB_MqttTelegram_Connect_V10, ST *)
(* @NESTEDCOMMENTS := 'Yes' *)
(* @PATH := '\/_Generic\/Mqtt\/Intern' *)
(* @OBJECTFLAGS := '0, 8' *)
(* @SYMFILEFLAGS := '2048' *)
FUNCTION_BLOCK FB_MqttTelegram_Connect_V10
VAR_IN_OUT
	stMqttSettings	: ST_MqttSettings;
END_VAR
VAR
	iState 				: INT := 0;
	idLength			: INT;
	iuLength			: INT;
	ipLength			: INT;
	ipos				: INT;
	stMqttTelegram		: ST_MqttTelegram;
	fbMqttEncodeLength	: FB_Mqtt_EncodeLength_V10;
	bLength1			: BYTE;
	bLength2			: BYTE;
	bLength3			: BYTE;
	bLength4			: BYTE;
	bLengthAmount		: BYTE;
END_VAR
VAR CONSTANT
	C_STARTUP		: INT := 0;
	C_BUILD_CONNECT	: INT := 100;
	C_SEND_WAIT		: INT := 110;
	C_IDLE			: INT := 500;
END_VAR
(* @END_DECLARATION := '0' *)
CASE iState OF
	C_STARTUP:
		IF
			NOT stMqttSettings.bDisconnect
			AND NOT stMqttSettings.bError
			AND stMqttSettings.bSocketConnection
			AND stMqttSettings.bActive
		THEN
			iState := C_IDLE;
		END_IF;

	(* build connect telegram *)
	C_BUILD_CONNECT:
		FC_Mqtt_ClearTelegram_V10(
			stMqttTelegram	:= stMqttTelegram,
			stMqttSettings	:= stMqttSettings
		);

		(* get client id length *)
		idLength := LEN(stMqttSettings.sMqttClientId);
		IF idLength < 1 THEN
			stMqttSettings.sMqttClientId := 'x';
			idLength := 1;
		END_IF;

		IF idLength > 23 THEN
			idLength := 23;
		END_IF;

		IF
			LEN(stMqttSettings.sMqttUserId) > 0
			AND LEN(stMqttSettings.sMqttPassword) > 0
		THEN
			iuLength := LEN(stMqttSettings.sMqttUserId)+2; (* 2 byte data length*)
			ipLength := LEN(stMqttSettings.sMqttPassword)+2; (* 2 byte data length*)
		ELSE
			iuLength := 0;
			ipLength := 0;
		END_IF

		(* Calculate length *)
		(* 10 byte header, 2 byte data length, data length, [user length + 2], [password length + 2]*)
		fbMqttEncodeLength(
			dwLength := 10 + 2 + INT_TO_BYTE(idLength) + INT_TO_BYTE(iuLength) + INT_TO_BYTE(ipLength),
			bLength1 => bLength1,
			bLength2 => bLength2,
			bLength3 => bLength3,
			bLength4 => bLength4,
			bAmount	 => bLengthAmount
		);

		(* MQTT Control Packet type *)
		stMqttTelegram.arMqttData[0] := 16;
		(* Remaining Length *)
		CASE bLengthAmount OF
			1:
				stMqttTelegram.arMqttData[1] := bLength1;

			2:
				stMqttTelegram.arMqttData[1] := bLength1;
				stMqttTelegram.arMqttData[2] := bLength2;

			3:
				stMqttTelegram.arMqttData[1] := bLength1;
				stMqttTelegram.arMqttData[2] := bLength2;
				stMqttTelegram.arMqttData[3] := bLength3;

			4:
				stMqttTelegram.arMqttData[1] := bLength1;
				stMqttTelegram.arMqttData[2] := bLength2;
				stMqttTelegram.arMqttData[3] := bLength3;
				stMqttTelegram.arMqttData[4] := bLength4;
		END_CASE;
		(* init position*)
		ipos := bLengthAmount;

		(* Length MSB *)
		stMqttTelegram.arMqttData[ipos+1] := 0;
		(* Length LSB *)
		stMqttTelegram.arMqttData[ipos+2] := 4;
		(* M *)
		stMqttTelegram.arMqttData[ipos+3] := 77;
		(* Q *)
		stMqttTelegram.arMqttData[ipos+4] := 81;
		(* T *)
		stMqttTelegram.arMqttData[ipos+5] := 84;
		(* T *)
		stMqttTelegram.arMqttData[ipos+6] := 84;
		(* Protocol Level *)
		stMqttTelegram.arMqttData[ipos+7] := 4;
		(* Connect Flags *)
		stMqttTelegram.arMqttData[ipos+8].1 := TRUE;
		stMqttTelegram.arMqttData[ipos+8].6 := (ipLength>2); (* more then 2 byte data length*)
		stMqttTelegram.arMqttData[ipos+8].7 := (iuLength>2); (* more then 2 byte data length*)
		(* Keep Alive MSB *)
		stMqttTelegram.arMqttData[ipos+9] := 0;
		(* Keep Alive LSB *)
		stMqttTelegram.arMqttData[ipos+10] := stMqttSettings.usKeepAliveTime;
		(* Data length MSB *)
		stMqttTelegram.arMqttData[ipos+11] := 0;
		(* Data length LSB *)
		stMqttTelegram.arMqttData[ipos+12] := INT_TO_BYTE(idLength);

		(* Client ID *)
		MEMCPY(
			destAddr	:= ADR(stMqttTelegram.arMqttData[ipos+13]),
		    srcAddr		:= ADR(stMqttSettings.sMqttClientId),
			n  			:= idLength
		);

		ipos := ipos+13+idLength;
		IF (iuLength > 2) THEN (* more then 2 byte data length*)
			(* Data length MSB *)
			stMqttTelegram.arMqttData[ipos] := 0;
			(* Data length LSB *)
			stMqttTelegram.arMqttData[ipos+1] := INT_TO_BYTE(iuLength-2);

			(* User ID *)
			MEMCPY(
				destAddr	:= ADR(stMqttTelegram.arMqttData[ipos+2]),
			    srcAddr		:= ADR(stMqttSettings.sMqttUserId),
				n  			:= iuLength-2
			);
			ipos := ipos+iuLength;
		END_IF

		IF (iuLength > 2) THEN (* more then 2 byte data length*)
			(* Data length MSB *)
			stMqttTelegram.arMqttData[ipos] := 0;
			(* Data length LSB *)
			stMqttTelegram.arMqttData[ipos+1] := INT_TO_BYTE(ipLength-2);

			(* Password *)
			MEMCPY(
				destAddr	:= ADR(stMqttTelegram.arMqttData[ipos+2]),
			    srcAddr		:= ADR(stMqttSettings.sMqttPassword),
				n  			:= ipLength-2
			);
			ipos := ipos+ipLength;
		END_IF

		stMqttTelegram.nDataLength 	:= ipos; (* 1 byte header, 1 byte remaining length *)
		iState 						:= C_SEND_WAIT;

	(* send telegram *)
	C_SEND_WAIT:
		IF stMqttSettings.stMqttSendTelegram.nDataLength = 0 THEN
			FC_Mqtt_CopyTelegram_V10(
				stMqttSrcTelegram	:= stMqttTelegram,
				stMqttDestTelegram	:= stMqttSettings.stMqttSendTelegram,
				stMqttSettings		:= stMqttSettings
			);

			stMqttSettings.bConnectPackageSent	:= TRUE;
			iState								:= C_IDLE;
		END_IF;

		IF
			NOT stMqttSettings.bActive
			OR NOT stMqttSettings.bSocketConnection
		THEN
			iState := C_STARTUP;
		END_IF;

	(* idle *)
	C_IDLE:
		IF
			NOT stMqttSettings.bDisconnect
			AND NOT stMqttSettings.bError
			AND NOT stMqttSettings.bConnected
			AND stMqttSettings.bSocketConnection
			AND NOT stMqttSettings.bConnectPackageSent
			AND stMqttSettings.bActive
		THEN
			iState := C_BUILD_CONNECT;
		END_IF;

		(* check received telegram *)
		IF
			stMqttSettings.bConnectPackageSent
			AND stMqttSettings.stMqttReceivedTelegram.nDataLength = 4
			AND stMqttSettings.stMqttReceivedTelegram.arMqttData[0] = 32
			AND stMqttSettings.stMqttReceivedTelegram.arMqttData[1] = 2
			AND (
				(* Session pressent or not, we ignore *)
				stMqttSettings.stMqttReceivedTelegram.arMqttData[2] = 1
				OR
				stMqttSettings.stMqttReceivedTelegram.arMqttData[2] = 0
			)
			AND stMqttSettings.stMqttReceivedTelegram.arMqttData[3] = 0
		THEN
			stMqttSettings.bConnected := TRUE;
			FC_Mqtt_ClearTelegram_V10(
				stMqttTelegram	:= stMqttSettings.stMqttReceivedTelegram,
				stMqttSettings	:= stMqttSettings
			);
		END_IF;

		(* error on connect *)
		IF
			stMqttSettings.bConnectPackageSent
			AND stMqttSettings.stMqttReceivedTelegram.nDataLength = 4
			AND stMqttSettings.stMqttReceivedTelegram.arMqttData[0] = 32
			AND stMqttSettings.stMqttReceivedTelegram.arMqttData[1] = 2
			AND stMqttSettings.stMqttReceivedTelegram.arMqttData[3] <> 0
		THEN
			stMqttSettings.bError := TRUE;
		END_IF;

		IF
			stMqttSettings.bDisconnect
			OR stMqttSettings.bError
			OR NOT stMqttSettings.bSocketConnection
			OR NOT stMqttSettings.bActive
		THEN
			iState := C_STARTUP;
		END_IF;

	ELSE
		iState := C_STARTUP;
END_CASE;


(*	END_FUNCTION_BLOCK	*)
END_FUNCTION_BLOCK

(* POU Intern/FB_Mqtt_EncodeLength_V10, ST *)
(* @NESTEDCOMMENTS := 'Yes' *)
(* @PATH := '\/_Generic\/Mqtt\/Intern' *)
(* @OBJECTFLAGS := '0, 8' *)
(* @SYMFILEFLAGS := '2048' *)
FUNCTION_BLOCK FB_Mqtt_EncodeLength_V10
VAR_INPUT
	dwLength	: DWORD;
END_VAR
VAR_OUTPUT
	bLength1	: BYTE := 0;
	bLength2	: BYTE := 0;
	bLength3	: BYTE := 0;
	bLength4	: BYTE := 0;
	bAmount		: BYTE := 0;
END_VAR
VAR
	dwWorkLength	: DWORD;
	dwCopyLength	: DWORD;
END_VAR
(* @END_DECLARATION := '0' *)
bAmount 		:= 1;
dwCopyLength	:= dwLength;

WHILE dwCopyLength > 0 DO
	dwWorkLength := dwCopyLength MOD 128;
	dwCopyLength := dwCopyLength / 128;

	IF dwCopyLength > 0 THEN
		dwWorkLength := dwWorkLength OR 128;
	END_IF;

	CASE bAmount OF
		1:
			bLength1 := DWORD_TO_BYTE(dwWorkLength);

		2:
			bLength2 := DWORD_TO_BYTE(dwWorkLength);

		3:
			bLength3 := DWORD_TO_BYTE(dwWorkLength);

		4:
			bLength4 := DWORD_TO_BYTE(dwWorkLength);

		ELSE
			;
	END_CASE;

	IF dwCopyLength > 0 THEN
		bAmount := bAmount + 1;
	END_IF;

	IF bAmount > 4 THEN
		(* hmm *)
		RETURN;
	END_IF;
END_WHILE;
(*
do
	encodedByte = X MOD 128
	X = X DIV 128

	// if there are more data to encode, set the top bit of this byte
	if ( X > 0 )
		encodedByte = encodedByte OR 128
	endif

	'output' encodedByte
while ( X > 0 )
*)

(*	END_FUNCTION_BLOCK	*)
END_FUNCTION_BLOCK

(* POU Intern/FC_Mqtt_ClearTelegram_V10, ST *)
(* @NESTEDCOMMENTS := 'Yes' *)
(* @PATH := '\/_Generic\/Mqtt\/Intern' *)
(* @OBJECTFLAGS := '0, 8' *)
(* @SYMFILEFLAGS := '2048' *)
FUNCTION FC_Mqtt_ClearTelegram_V10 : BOOL
VAR_IN_OUT
	stMqttTelegram	: ST_MqttTelegram;
	stMqttSettings	: ST_MqttSettings;
END_VAR
VAR
END_VAR
(* @END_DECLARATION := '0' *)
MEMSET(
	destAddr	:= ADR(stMqttTelegram.arMqttData),
	fillByte  	:= 0,
	n			:= stMqttSettings.iTelegramSize
);

stMqttTelegram.nDataLength := 0;

(*	END_FUNCTION	*)
END_FUNCTION

(* POU Intern/FC_Mqtt_CopyTelegram_V10, ST *)
(* @NESTEDCOMMENTS := 'Yes' *)
(* @PATH := '\/_Generic\/Mqtt\/Intern' *)
(* @OBJECTFLAGS := '0, 8' *)
(* @SYMFILEFLAGS := '2048' *)
FUNCTION FC_Mqtt_CopyTelegram_V10 : BOOL
VAR_IN_OUT
	stMqttSrcTelegram	: ST_MqttTelegram;
	stMqttDestTelegram	: ST_MqttTelegram;
	stMqttSettings		: ST_MqttSettings;
END_VAR
VAR
END_VAR
(* @END_DECLARATION := '0' *)
MEMCPY(
	destAddr	:= ADR(stMqttDestTelegram.arMqttData),
    srcAddr		:= ADR(stMqttSrcTelegram.arMqttData),
	n  			:= stMqttSettings.iTelegramSize
);

stMqttDestTelegram.nDataLength := stMqttSrcTelegram.nDataLength;

(*	END_FUNCTION	*)
END_FUNCTION

(* POU Intern/FB_MqttTelegram_PingReq_V10, ST *)
(* @NESTEDCOMMENTS := 'Yes' *)
(* @PATH := '\/_Generic\/Mqtt\/Intern' *)
(* @OBJECTFLAGS := '0, 8' *)
(* @SYMFILEFLAGS := '2048' *)
FUNCTION_BLOCK FB_MqttTelegram_PingReq_V10
VAR_IN_OUT
	stMqttSettings	: ST_MqttSettings;
END_VAR
VAR
	iState 				: INT := 0;
	bMustSend			: BOOL := FALSE;
	bPingReqSent		: BOOL := FALSE;
	stMqttTelegram		: ST_MqttTelegram;
END_VAR
VAR CONSTANT
	C_STARTUP		: INT := 0;
	C_BUILD_PING	: INT := 100;
	C_SEND_WAIT		: INT := 110;
	C_IDLE			: INT := 500;
END_VAR
(* @END_DECLARATION := '0' *)
CASE iState OF
	C_STARTUP:
		bPingReqSent := FALSE;

		IF stMqttSettings.bValidConnection THEN
			iState := C_IDLE;
		END_IF;

	(* build pingreq telegram *)
	C_BUILD_PING:
		FC_Mqtt_ClearTelegram_V10(
			stMqttTelegram	:= stMqttTelegram,
			stMqttSettings	:= stMqttSettings
		);

		(* MQTT Control Packet type *)
		stMqttTelegram.arMqttData[0] := 192;
		(* Remaining Length *)
		stMqttTelegram.arMqttData[1] := 0;

		stMqttTelegram.nDataLength := 2;

		iState := C_SEND_WAIT;

	(* send telegram *)
	C_SEND_WAIT:
		IF stMqttSettings.stMqttSendTelegram.nDataLength = 0 THEN
			FC_Mqtt_CopyTelegram_V10(
				stMqttSrcTelegram	:= stMqttTelegram,
				stMqttDestTelegram	:= stMqttSettings.stMqttSendTelegram,
				stMqttSettings		:= stMqttSettings
			);

			bPingReqSent	:= TRUE;
			iState			:= C_IDLE;
		END_IF;

		IF NOT stMqttSettings.bValidConnection THEN
			iState := C_STARTUP;
		END_IF;

	(* idle *)
	C_IDLE:
		bMustSend := FALSE;

		IF stMqttSettings.usKeepAliveTime > 0 THEN
			bMustSend := stMqttSettings.tonSendPingReq.Q;
		END_IF;

		IF
			stMqttSettings.bValidConnection
			AND bMustSend
			AND NOT bPingReqSent
		THEN
			iState := C_BUILD_PING;
		END_IF;

		(* Check received telegram *)
		IF
			bPingReqSent
			AND stMqttSettings.stMqttReceivedTelegram.nDataLength = 2
			AND stMqttSettings.stMqttReceivedTelegram.arMqttData[0] = 208
			AND stMqttSettings.stMqttReceivedTelegram.arMqttData[1] = 0
		THEN
			FC_Mqtt_ClearTelegram_V10(
				stMqttTelegram	:= stMqttSettings.stMqttReceivedTelegram,
				stMqttSettings	:= stMqttSettings
			);
			bPingReqSent := FALSE;
		END_IF;

		IF NOT stMqttSettings.bValidConnection THEN
			iState := C_STARTUP;
		END_IF;

	ELSE
		iState := C_STARTUP;
END_CASE;

(*	END_FUNCTION_BLOCK	*)
END_FUNCTION_BLOCK

(* POU Intern/FB_Mqtt_Send_V10, ST *)
(* @NESTEDCOMMENTS := 'Yes' *)
(* @PATH := '\/_Generic\/Mqtt\/Intern' *)
(* @OBJECTFLAGS := '0, 8' *)
(* @SYMFILEFLAGS := '2048' *)
FUNCTION_BLOCK FB_Mqtt_Send_V10
VAR_OUTPUT
	bBusy	: BOOL := FALSE;
END_VAR
VAR_IN_OUT
	stMqttSettings	: ST_MqttSettings;
END_VAR
VAR
	fbSocketSend 	: FB_SocketSend;
	tPingReq		: TIME;
	iState 			: INT := 0;
	stSendTelegram	: ST_MqttTelegram;
END_VAR
VAR CONSTANT
	C_STARTUP		: INT := 0;
	C_SEND			: INT := 100;
	C_SEND_WAIT		: INT := 110;
	C_IDLE			: INT := 500;
END_VAR
(* @END_DECLARATION := '0' *)
CASE iState OF
	C_STARTUP:
		bBusy := FALSE;

		stMqttSettings.tonSendPingReq(
			in := FALSE
		);

		IF
			NOT stMqttSettings.bDisconnect
			AND NOT stMqttSettings.bError
			AND stMqttSettings.bSocketConnection
		THEN
			iState := C_IDLE;
		END_IF;

	(* send mqtt telegram *)
	C_SEND:
		bBusy := TRUE;

		(* copy send telegram *)
		FC_Mqtt_CopyTelegram_V10(
			stMqttSrcTelegram	:= stMqttSettings.stMqttSendTelegram,
			stMqttDestTelegram	:= stSendTelegram,
			stMqttSettings		:= stMqttSettings
		);

		(* start send *)
		fbSocketSend(
			bExecute := FALSE
		);

		fbSocketSend(
			sSrvNetId	:= '',
			hSocket		:= stMqttSettings.hSocket,
			cbLen		:= stSendTelegram.nDataLength,
			pSrc		:= ADR(stSendTelegram.arMqttData),
			bExecute 	:= TRUE
		);

		iState := C_SEND_WAIT;

	(* wait send done *)
	C_SEND_WAIT:
		fbSocketSend(
			bExecute := FALSE
		);

		IF
			NOT fbSocketSend.bBusy
			AND NOT fbSocketSend.bError
		THEN
			(* copy last telegram *)
			FC_Mqtt_CopyTelegram_V10(
				stMqttSrcTelegram	:= stMqttSettings.stMqttSendTelegram,
				stMqttDestTelegram	:= stMqttSettings.stMqttLastSendTelegram,
				stMqttSettings		:= stMqttSettings
			);

			(* clear send buffer *)
			FC_Mqtt_ClearTelegram_V10(
				stMqttTelegram 	:= stMqttSettings.stMqttSendTelegram,
				stMqttSettings	:= stMqttSettings
			);

			iState	:= C_IDLE;
			bBusy	:= FALSE;
		END_IF;

		IF stMqttSettings.usKeepAliveTime > 0 THEN
			tPingReq := DWORD_TO_TIME(USINT_TO_DWORD(stMqttSettings.usKeepAliveTime) * 1000 - 5000);

			stMqttSettings.tonSendPingReq(
				in := FALSE
			);

			stMqttSettings.tonSendPingReq(
				in := TRUE,
				pt := tPingReq
			);
		END_IF;

		IF fbSocketSend.bError THEN
			iState 					:= C_STARTUP;
			stMqttSettings.bError	:= TRUE;
		END_IF;

		IF
			NOT stMqttSettings.bActive
			OR NOT stMqttSettings.bSocketConnection
		THEN
			iState := C_STARTUP;
		END_IF;

	(* idle *)
	C_IDLE:
		IF stMqttSettings.usKeepAliveTime > 0 THEN
			stMqttSettings.tonSendPingReq(
				in := stMqttSettings.bConnected
			);
		ELSE
			stMqttSettings.tonSendPingReq(
				in := FALSE
			);
		END_IF;

		IF
			stMqttSettings.stMqttSendTelegram.nDataLength > 0
			AND NOT stMqttSettings.bDisconnect
			AND NOT stMqttSettings.bError
			AND stMqttSettings.bSocketConnection
			AND NOT bBusy
		THEN
			iState := C_SEND;
		END_IF;

		IF
			stMqttSettings.bDisconnect
			OR stMqttSettings.bError
			OR NOT stMqttSettings.bSocketConnection
		THEN
			iState := C_STARTUP;
		END_IF;

		(* ensure at least 1 cycle pause *)
		(* bBusy := FALSE; *)

	ELSE
		iState := C_STARTUP;
END_CASE;

(*	END_FUNCTION_BLOCK	*)
END_FUNCTION_BLOCK

(* POU Intern/FB_Mqtt_Receive_V10, ST *)
(* @NESTEDCOMMENTS := 'Yes' *)
(* @PATH := '\/_Generic\/Mqtt\/Intern' *)
(* @OBJECTFLAGS := '0, 8' *)
(* @SYMFILEFLAGS := '2048' *)
FUNCTION_BLOCK FB_Mqtt_Receive_V10
VAR_OUTPUT
	bBusy	: BOOL := FALSE;
END_VAR
VAR_IN_OUT
	stMqttSettings	: ST_MqttSettings;
END_VAR
VAR
	fbSocketReceive		: FB_SocketReceive;
	fbMqttDecodeLength	: FB_Mqtt_DecodeLength_V10;
	stReceiveBuffer		: ST_MqttTelegram;

	iState 			: INT := 0;
	iLengthPosition	: INT := 0;
	index			: INT := 0;
	dwDataLength	: DWORD := 0;
	wTopicLength	: WORD := 0;
	dwValueLength	: DWORD := 0;
END_VAR
VAR CONSTANT
	C_STARTUP				: INT := 0;
	C_RECEIVE_HEADER		: INT := 100;
	C_RECEIVE_HEADER_WAIT	: INT := 110;
	C_RECEIVE_LENGTH		: INT := 120;
	C_RECEIVE_LENGTH_WAIT	: INT := 130;
	C_RECEIVE_DATA			: INT := 200;
	C_RECEIVE_DATA_WAIT		: INT := 210;
	C_IDLE					: INT := 500;
END_VAR

(* @END_DECLARATION := '0' *)
CASE iState OF
	C_STARTUP:
		bBusy 			:= FALSE;
		iLengthPosition	:= 0;
		index			:= 0;
		dwDataLength	:= 0;
		wTopicLength	:= 0;
		dwValueLength	:= 0;
		ClearReceivedPublishTelegram();

		IF
			NOT stMqttSettings.bDisconnect
			AND NOT stMqttSettings.bError
			AND stMqttSettings.bSocketConnection
		THEN
			iState := C_IDLE;
		END_IF;

	(* start receive header *)
	C_RECEIVE_HEADER:
		bBusy := TRUE;
		ClearReceivedPublishTelegram();

		fbSocketReceive(
			bExecute := FALSE
		);

		fbSocketReceive(
			sSrvNetId	:= '',
			hSocket		:= stMqttSettings.hSocket,
			cbLen		:= 2,
			pDest		:= ADR(stReceiveBuffer.arMqttData),
			bExecute 	:= TRUE
		);

		iState := C_RECEIVE_HEADER_WAIT;

	(* wait for header with length *)
	C_RECEIVE_HEADER_WAIT:
		fbSocketReceive(
			bExecute := FALSE
		);

		IF
			NOT fbSocketReceive.bBusy
			AND NOT fbSocketReceive.bError
			AND fbSocketReceive.nRecBytes = 2
		THEN
			iLengthPosition	:= 0;
			stMqttSettings.stMqttReceivedTelegram.arMqttData[0] := stReceiveBuffer.arMqttData[0];
			stMqttSettings.stMqttReceivedTelegram.arMqttData[1] := stReceiveBuffer.arMqttData[1];

			IF stMqttSettings.stMqttReceivedTelegram.arMqttData[1].7 = 1 THEN
				(* payload longer then 127 byte *)
				iLengthPosition := iLengthPosition + 1;
				iState			:= C_RECEIVE_LENGTH;
			ELSE
				IF stMqttSettings.stMqttReceivedTelegram.arMqttData[1] = 0 THEN
					(* no payload received *)
					stMqttSettings.stMqttReceivedTelegram.nDataLength := 2;

					(* copy last telegram *)
					FC_Mqtt_CopyTelegram_V10(
						stMqttSrcTelegram	:= stMqttSettings.stMqttReceivedTelegram,
						stMqttDestTelegram	:= stMqttSettings.stMqttLastReceivedTelegram,
						stMqttSettings		:= stMqttSettings
					);

					iState	:= C_IDLE;
					bBusy 	:= FALSE;
				ELSE
					iState := C_RECEIVE_DATA;
				END_IF;
			END_IF;
		END_IF;

		IF fbSocketReceive.bError THEN
			iState 					:= C_STARTUP;
			stMqttSettings.bError	:= TRUE;
		END_IF;

		IF fbSocketReceive.nRecBytes = 0 THEN
			iState	:= C_IDLE;
			bBusy	:= FALSE;
		END_IF;

		IF
			NOT stMqttSettings.bActive
			OR NOT stMqttSettings.bSocketConnection
		THEN
			iState := C_STARTUP;
		END_IF;

	(* read next remaining length *)
	C_RECEIVE_LENGTH:
		fbSocketReceive(
			bExecute := FALSE
		);

		fbSocketReceive(
			sSrvNetId	:= '',
			hSocket		:= stMqttSettings.hSocket,
			cbLen		:= 1,
			pDest		:= ADR(stReceiveBuffer.arMqttData),
			bExecute 	:= TRUE
		);

		iState := C_RECEIVE_LENGTH_WAIT;

	(* wait for remaining length *)
	C_RECEIVE_LENGTH_WAIT:
		fbSocketReceive(
			bExecute := FALSE
		);

		IF
			NOT fbSocketReceive.bBusy
			AND NOT fbSocketReceive.bError
			AND fbSocketReceive.nRecBytes = 1
		THEN
			stMqttSettings.stMqttReceivedTelegram.arMqttData[1 + iLengthPosition] := stReceiveBuffer.arMqttData[0];

			IF stMqttSettings.stMqttReceivedTelegram.arMqttData[1 + iLengthPosition].7 = 1 THEN
				(* read next length byte *)
				iLengthPosition := iLengthPosition + 1;
				iState			:= C_RECEIVE_LENGTH;

				(* Not more the 4 length bytes *)
				IF iLengthPosition > 4 THEN
					iState 					:= C_STARTUP;
					stMqttSettings.bError	:= TRUE;
				END_IF;
			ELSE
				iState := C_RECEIVE_DATA;
			END_IF;
		END_IF;

		IF fbSocketReceive.bError THEN
			iState 					:= C_STARTUP;
			stMqttSettings.bError	:= TRUE;
		END_IF;

		IF
			NOT stMqttSettings.bActive
			OR NOT stMqttSettings.bSocketConnection
		THEN
			iState := C_STARTUP;
		END_IF;

	(* receive remaining data *)
	C_RECEIVE_DATA:
		fbMqttDecodeLength(
			stMqttTelegram	:= stMqttSettings.stMqttReceivedTelegram,
			dwLength		=> dwDataLength
		);

		fbSocketReceive(
			bExecute := FALSE
		);

		fbSocketReceive(
			sSrvNetId	:= '',
			hSocket		:= stMqttSettings.hSocket,
			cbLen		:= dwDataLength,
			pDest		:= ADR(stReceiveBuffer.arMqttData),
			bExecute 	:= TRUE
		);

		iState := C_RECEIVE_DATA_WAIT;

	(* receive *)
	C_RECEIVE_DATA_WAIT:
		fbSocketReceive(
			bExecute := FALSE
		);

		IF
			NOT fbSocketReceive.bBusy
			AND NOT fbSocketReceive.bError
			AND fbSocketReceive.nRecBytes > 0
		THEN
			MEMCPY(
				destAddr	:= ADR(stMqttSettings.stMqttReceivedTelegram.arMqttData[2 + iLengthPosition]),
			    srcAddr		:= ADR(stReceiveBuffer.arMqttData),
				n  			:= fbSocketReceive.nRecBytes
			);
			stMqttSettings.stMqttReceivedTelegram.nDataLength := 2 + iLengthPosition + fbSocketReceive.nRecBytes;

			(* copy last telegram *)
			FC_Mqtt_CopyTelegram_V10(
				stMqttSrcTelegram	:= stMqttSettings.stMqttReceivedTelegram,
				stMqttDestTelegram	:= stMqttSettings.stMqttLastReceivedTelegram,
				stMqttSettings		:= stMqttSettings
			);

			(* check for publish *)
			IF (stMqttSettings.stMqttReceivedTelegram.arMqttData[0] AND 48) = 48 THEN
				ClearReceivedPublishTelegram();

				(* Length MSB/LSB Topic *)
				wTopicLength :=
						SHL(BYTE_TO_WORD(stMqttSettings.stMqttReceivedTelegram.arMqttData[2 + iLengthPosition + 1]), 8) +
						BYTE_TO_WORD(stMqttSettings.stMqttReceivedTelegram.arMqttData[1 + iLengthPosition + 1]);
				wTopicLength := BE16_TO_HOST(wTopicLength);

				(* Copy topic *)
				MEMCPY(
					destAddr	:= ADR(stMqttSettings.stMqttReceivedPublishTelegram.sTopic),
				    srcAddr		:= ADR(stMqttSettings.stMqttReceivedTelegram.arMqttData[3 + iLengthPosition + 1]),
					n  			:= wTopicLength
				);

				(* Copy value *)
				(* value length = remaining data length - length topic value - 2 byte topic length *)
				dwValueLength := dwDataLength - wTopicLength - 2;

				MEMCPY(
					destAddr	:= ADR(stMqttSettings.stMqttReceivedPublishTelegram.sValue),
				    srcAddr		:= ADR(stMqttSettings.stMqttReceivedTelegram.arMqttData[3 + iLengthPosition + 1 + wTopicLength]),
					n  			:= dwValueLength
				);

				stMqttSettings.stMqttReceivedPublishTelegram.bHasData := TRUE;
			END_IF;

			iState	:= C_IDLE;
			bBusy	:= FALSE;
		END_IF;

		IF fbSocketReceive.bError THEN
			iState 					:= C_STARTUP;
			stMqttSettings.bError	:= TRUE;
		END_IF;

		IF
			NOT stMqttSettings.bActive
			OR NOT stMqttSettings.bSocketConnection
		THEN
			iState := C_STARTUP;
		END_IF;

	(* idle *)
	C_IDLE:
		IF
			NOT stMqttSettings.bDisconnect
			AND NOT stMqttSettings.bError
			AND stMqttSettings.bSocketConnection
			AND NOT bBusy
		THEN
			iState := C_RECEIVE_HEADER;
		END_IF;

		IF
			stMqttSettings.bDisconnect
			OR stMqttSettings.bError
			OR NOT stMqttSettings.bSocketConnection
		THEN
			iState := C_STARTUP;
		END_IF;

		(* ensure at least 1 cycle pause *)
		(* bBusy := FALSE; *)

	ELSE
		iState := C_STARTUP;
END_CASE;

(*	END_FUNCTION_BLOCK	*)
END_FUNCTION_BLOCK
ACTION ClearReceivedPublishTelegram:
MEMSET(
	destAddr	:= ADR(stMqttSettings.stMqttReceivedPublishTelegram.sTopic),
	fillByte  	:= 0,
	n			:= 255
);
stMqttSettings.stMqttReceivedPublishTelegram.sTopic := '';

MEMSET(
	destAddr	:= ADR(stMqttSettings.stMqttReceivedPublishTelegram.sValue),
	fillByte  	:= 0,
	n			:= 255
);
stMqttSettings.stMqttReceivedPublishTelegram.sValue := '';

stMqttSettings.stMqttReceivedPublishTelegram.bHasData := FALSE;
END_ACTION

(* POU Intern/FB_Mqtt_DecodeLength_V10, ST *)
(* @NESTEDCOMMENTS := 'Yes' *)
(* @PATH := '\/_Generic\/Mqtt\/Intern' *)
(* @OBJECTFLAGS := '0, 8' *)
(* @SYMFILEFLAGS := '2048' *)
FUNCTION_BLOCK FB_Mqtt_DecodeLength_V10
VAR_INPUT
	stMqttTelegram : ST_MqttTelegram;
END_VAR
VAR_OUTPUT
	dwLength	: DWORD;
	bAmount		: BYTE;
END_VAR
VAR
	index			: INT;
	diMultiplier	: DINT;
	dwValue			: DWORD;
END_VAR
(* @END_DECLARATION := '0' *)
index			:= 0;
diMultiplier	:= 1;
dwValue			:= 0;

REPEAT
	index := index + 1;

	dwValue := dwValue + (stMqttTelegram.arMqttData[index] AND 127) * diMultiplier;
	diMultiplier := diMultiplier * 128;

	IF diMultiplier > 128*128*128 THEN
		dwLength	:= 0;
		bAmount		:= 0;
		RETURN;
	END_IF;
UNTIL stMqttTelegram.arMqttData[index].7 = 0
END_REPEAT;

dwLength	:= dwValue;
bAmount		:= INT_TO_BYTE(index);

(*
multiplier = 1
value = 0

do
	encodedByte = 'next byte from stream'
	value += (encodedByte AND 127) * multiplier
	multiplier *= 128

	if (multiplier > 128*128*128)
		throw Error(Malformed Remaining Length)
while ((encodedByte AND 128) != 0)

*)

(*	END_FUNCTION_BLOCK	*)
END_FUNCTION_BLOCK

